KUKA KRL program: MyProgram_025().src

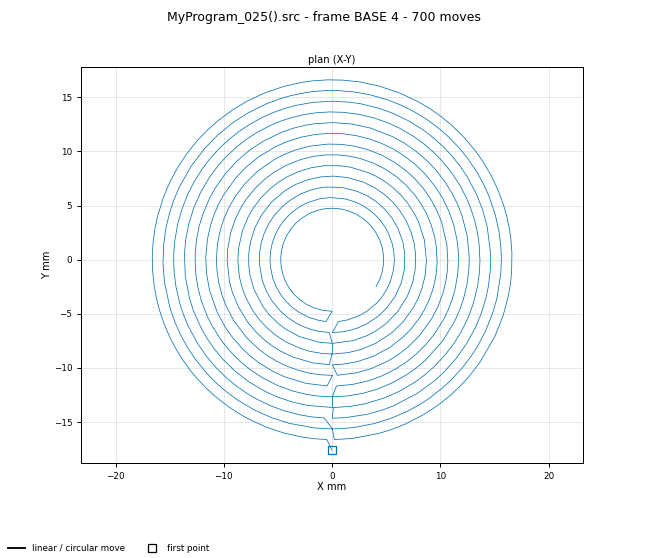
[picture p0: tool path of MyProgram_025().src in frame BASE 4, 700 of 700 moves have a stored position in this frame; points joined in program order, loops and branches not executed]
&ACCESS RVP
&REL 1
&PARAM TEMPLATE = C:\KRC\Roboter\Template\vorgabe
&PARAM EDITMASK = *
DEF MyProgram_025()
; ---- Setting reference (Base) ----
$BASE = BASE_DATA[4]

; --------------------------
; ---- Setting tool (TCP) ----
$TOOL = TOOL_DATA[3]
; --------------------------

$VEL.CP = VEL_APROX_PRINT
Startdeposition()
$VEL.CP = VEL_PRINT
LIN {X -0.0079,Y -17.5993,Z 57,A -96.7088,B 24.8277,C -3.0276,E1 25.0016,E2 -540.8331} C_DIS
Enddeposition()
LIN {X -0.0079,Y -17.5993,Z 57,A -96.7088,B 24.8277,C -3.0276,E1 25.0016,E2 -540.8331} C_DIS
Startdeposition()
$VEL.CP = VEL_PRINT
LIN {X -0.4966,Y -16.6086,Z 57,A -99.8681,B 24.8268,C -3.0359,E1 24.9929,E2 -537.6934} C_DIS
LIN {X -1.6135,Y -16.537,Z 57,A -103.5164,B 24.8266,C -3.0371,E1 24.9827,E2 -534.0464} C_DIS
LIN {X -2.8447,Y -16.3711,Z 57,A -108.4437,B 24.8269,C -3.0348,E1 24.9691,E2 -529.1094} C_DIS
LIN {X -4.4562,Y -16.0071,Z 57,A -114.0393,B 24.8265,C -3.0384,E1 24.9539,E2 -523.5144} C_DIS
LIN {X -6.0086,Y -15.4911,Z 57,A -120.3212,B 24.8262,C -3.0403,E1 24.9374,E2 -517.2245} C_DIS
LIN {X -7.613,Y -14.7693,Z 57,A -125.0534,B 24.8248,C -3.0528,E1 24.9255,E2 -512.51} C_DIS
LIN {X -8.4976,Y -14.2789,Z 57,A -129.0744,B 24.8245,C -3.0554,E1 24.9158,E2 -508.4833} C_DIS
LIN {X -9.6445,Y -13.5307,Z 57,A -134.1192,B 24.8238,C -3.0616,E1 24.9042,E2 -503.4363} C_DIS
LIN {X -10.8321,Y -12.6002,Z 57,A -138.7295,B 24.8225,C -3.073,E1 24.8942,E2 -498.8359} C_DIS
LIN {X -11.5957,Y -11.9014,Z 57,A -142.6614,B 24.8218,C -3.0788,E1 24.8862,E2 -494.9017} C_DIS
LIN {X -12.5279,Y -10.9156,Z 57,A -146.9241,B 24.8205,C -3.0901,E1 24.8782,E2 -490.6474} C_DIS
LIN {X -13.1346,Y -10.1775,Z 57,A -150.5821,B 24.8197,C -3.0966,E1 24.8718,E2 -486.9877} C_DIS
LIN {X -13.8252,Y -9.2175,Z 57,A -154.4634,B 24.8185,C -3.107,E1 24.8656,E2 -483.1122} C_DIS
LIN {X -14.4131,Y -8.2642,Z 57,A -158.3118,B 24.8173,C -3.117,E1 24.8601,E2 -479.2678} C_DIS
LIN {X -15.0085,Y -7.1299,Z 57,A -163.0011,B 24.816,C -3.128,E1 24.8542,E2 -474.5798} C_DIS
LIN {X -15.5303,Y -5.9078,Z 57,A -167.967,B 24.8146,C -3.1399,E1 24.849,E2 -469.6147} C_DIS
LIN {X -15.9455,Y -4.6722,Z 57,A -172.1158,B 24.813,C -3.1538,E1 24.8455,E2 -465.4753} C_DIS
LIN {X -16.2237,Y -3.5903,Z 57,A -175.9774,B 24.8116,C -3.1652,E1 24.843,E2 -461.6184} C_DIS
LIN {X -16.4274,Y -2.4984,Z 57,A -179.9383,B 24.8103,C -3.1765,E1 24.8412,E2 -457.6611} C_DIS
LIN {X -16.5879,Y -0.9632,Z 57,A 174.764,B 24.8083,C -3.1929,E1 24.8399,E2 -452.3709} C_DIS
LIN {X -16.6147,Y 0.2389,Z 57,A 170.0951,B 24.8069,C -3.2046,E1 24.8399,E2 -447.702} C_DIS
LIN {X -16.5377,Y 1.6093,Z 57,A 166.0881,B 24.8049,C -3.2209,E1 24.8407,E2 -443.71} C_DIS
LIN {X -16.379,Y 2.7981,Z 57,A 162.1452,B 24.8033,C -3.2342,E1 24.8423,E2 -439.7753} C_DIS
LIN {X -16.1488,Y 3.9123,Z 57,A 156.9096,B 24.8021,C -3.2434,E1 24.8455,E2 -434.531} C_DIS
LIN {X -15.6026,Y 5.7141,Z 57,A 150.5557,B 24.7997,C -3.2632,E1 24.8512,E2 -428.1884} C_DIS
LIN {X -15.0536,Y 7.0344,Z 57,A 145.873,B 24.7979,C -3.2781,E1 24.8565,E2 -423.5158} C_DIS
LIN {X -14.2835,Y 8.4901,Z 57,A 139.9499,B 24.7959,C -3.2935,E1 24.8645,E2 -417.5984} C_DIS
LIN {X -13.4224,Y 9.7912,Z 57,A 135.2799,B 24.7939,C -3.3097,E1 24.8719,E2 -412.9442} C_DIS
LIN {X -12.4942,Y 10.9541,Z 57,A 130.3829,B 24.7922,C -3.3233,E1 24.8806,E2 -408.057} C_DIS
LIN {X -11.6781,Y 11.8204,Z 57,A 125.1708,B 24.7914,C -3.3297,E1 24.8907,E2 -402.838} C_DIS
LIN {X -10.5248,Y 12.858,Z 57,A 120.5872,B 24.7896,C -3.3437,E1 24.9004,E2 -398.27} C_DIS
LIN {X -9.1848,Y 13.847,Z 57,A 114.2189,B 24.7885,C -3.3529,E1 24.9149,E2 -391.9016} C_DIS
LIN {X -7.7571,Y 14.6943,Z 57,A 108.4775,B 24.7873,C -3.3625,E1 24.9288,E2 -386.1666} C_DIS
LIN {X -6.1672,Y 15.429,Z 57,A 102.3711,B 24.7862,C -3.3708,E1 24.9445,E2 -380.0655} C_DIS
LIN {X -4.4893,Y 15.9979,Z 57,A 96.3662,B 24.7853,C -3.378,E1 24.9604,E2 -374.0674} C_DIS
LIN {X -2.884,Y 16.364,Z 57,A 90.9322,B 24.7846,C -3.3837,E1 24.9753,E2 -368.6406} C_DIS
LIN {X -1.7423,Y 16.5244,Z 57,A 86.9351,B 24.7843,C -3.3859,E1 24.9863,E2 -364.6459} C_DIS
LIN {X -0.406,Y 16.6112,Z 57,A 82.7039,B 24.7838,C -3.3894,E1 24.9981,E2 -360.422} C_DIS
LIN {X 0.9946,Y 16.5858,Z 57,A 77.1037,B 24.7843,C -3.3858,E1 25.0138,E2 -354.8146} C_DIS
LIN {X 2.6236,Y 16.4076,Z 57,A 71.2834,B 24.7846,C -3.3836,E1 25.0299,E2 -348.9939} C_DIS
LIN {X 4.2635,Y 16.0596,Z 57,A 65.3163,B 24.7851,C -3.3793,E1 25.046,E2 -343.0255} C_DIS
LIN {X 6.1988,Y 15.4163,Z 57,A 58.4682,B 24.7858,C -3.3743,E1 25.064,E2 -336.1796} C_DIS
LIN {X 8.0336,Y 14.5452,Z 57,A 52.1599,B 24.7863,C -3.3702,E1 25.0797,E2 -329.8788} C_DIS
LIN {X 8.9547,Y 13.9969,Z 57,A 48.0765,B 24.7873,C -3.3622,E1 25.0894,E2 -325.7892} C_DIS
LIN {X 10.1005,Y 13.1939,Z 57,A 43.99,B 24.7877,C -3.3593,E1 25.0986,E2 -321.7103} C_DIS
LIN {X 10.9536,Y 12.4947,Z 57,A 39.5699,B 24.7891,C -3.3478,E1 25.1081,E2 -317.28} C_DIS
LIN {X 12.0575,Y 11.4333,Z 57,A 34.1471,B 24.7906,C -3.3359,E1 25.1187,E2 -311.8518} C_DIS
LIN {X 13.1886,Y 10.1074,Z 57,A 29.0536,B 24.7915,C -3.3292,E1 25.1278,E2 -306.766} C_DIS
LIN {X 13.9189,Y 9.0749,Z 57,A 23.824,B 24.7937,C -3.3117,E1 25.136,E2 -301.5208} C_DIS
LIN {X 14.6967,Y 7.7524,Z 57,A 18.6399,B 24.7953,C -3.2987,E1 25.1431,E2 -296.3328} C_DIS
LIN {X 15.312,Y 6.4523,Z 57,A 14.2767,B 24.7964,C -3.2899,E1 25.1481,E2 -291.9724} C_DIS
LIN {X 15.8274,Y 5.0576,Z 57,A 8.8948,B 24.7985,C -3.2732,E1 25.1531,E2 -286.581} C_DIS
LIN {X 16.1435,Y 3.9343,Z 57,A 4.9444,B 24.7999,C -3.2619,E1 25.1559,E2 -282.6266} C_DIS
LIN {X 16.3628,Y 2.8911,Z 57,A 1.4471,B 24.801,C -3.2523,E1 25.1577,E2 -279.127} C_DIS
LIN {X 16.5081,Y 1.8912,Z 57,A -2.0127,B 24.8023,C -3.2418,E1 25.159,E2 -275.6629} C_DIS
LIN {X 16.6046,Y 0.6127,Z 57,A -7.3278,B 24.8049,C -3.2206,E1 25.1598,E2 -270.3291} C_DIS
LIN {X 16.572,Y -1.2047,Z 57,A -12.6063,B 24.8063,C -3.2095,E1 25.1592,E2 -265.0555} C_DIS
LIN {X 16.4651,Y -2.2352,Z 57,A -16.4567,B 24.8079,C -3.196,E1 25.1579,E2 -261.1959} C_DIS
LIN {X 16.2794,Y -3.328,Z 57,A -20.8494,B 24.8099,C -3.1794,E1 25.1555,E2 -256.7894} C_DIS
LIN {X 15.7843,Y -5.1905,Z 57,A -26.4474,B 24.8113,C -3.1679,E1 25.1512,E2 -251.1963} C_DIS
LIN {X 15.0304,Y -7.083,Z 57,A -35.0616,B 24.8153,C -3.1341,E1 25.1417,E2 -242.5491} C_DIS
LIN {X 13.6579,Y -9.4636,Z 57,A -44.0363,B 24.8179,C -3.1121,E1 25.1283,E2 -233.5676} C_DIS
LIN {X 12.6386,Y -10.7872,Z 57,A -48.808,B 24.8187,C -3.1052,E1 25.12,E2 -228.8016} C_DIS
LIN {X 11.8964,Y -11.6005,Z 57,A -52.9805,B 24.8201,C -3.0931,E1 25.1119,E2 -224.6186} C_DIS
LIN {X 10.9268,Y -12.5181,Z 57,A -57.6642,B 24.8214,C -3.0822,E1 25.1022,E2 -219.9277} C_DIS
LIN {X 9.7819,Y -13.4314,Z 57,A -62.0262,B 24.822,C -3.0768,E1 25.0925,E2 -215.569} C_DIS
LIN {X 8.4724,Y -14.2939,Z 57,A -68.8986,B 24.8244,C -3.0564,E1 25.0762,E2 -208.6699} C_DIS
LIN {X 6.7566,Y -15.18,Z 57,A -73.9115,B 24.8243,C -3.0574,E1 25.0636,E2 -203.6725} C_DIS
LIN {X 5.5988,Y -15.6442,Z 57,A -79.1554,B 24.8257,C -3.0455,E1 25.0499,E2 -198.4115} C_DIS
LIN {X 4.3439,Y -16.0381,Z 57,A -84.2086,B 24.8266,C -3.0374,E1 25.0363,E2 -193.3474} C_DIS
LIN {X 1.8661,Y -16.5109,Z 57,A -91.9923,B 24.8266,C -3.0367,E1 25.0148,E2 -185.5698} C_DIS
LIN {X 0.2013,Y -16.6148,Z 57,A -97.7093,B 24.8269,C -3.0348,E1 24.9989,E2 -179.85} C_DIS
LIN {X 0.2013,Y -16.6148,Z 57,A -97.7093,B 24.8269,C -3.0348,E1 24.9989,E2 -179.85} C_DIS
Enddeposition()
LIN {X 0.0206,Y -15.6269,Z 57,A -98.3842,B 24.8249,C -3.0519,E1 24.9971,E2 -179.2158} C_DIS
Startdeposition()
$VEL.CP = VEL_PRINT
LIN {X 0.9435,Y -15.599,Z 57,A -93.051,B 24.8236,C -3.0635,E1 25.0121,E2 -184.5756} C_DIS
LIN {X 2.0952,Y -15.4866,Z 57,A -87.9065,B 24.8227,C -3.0713,E1 25.0264,E2 -189.7346} C_DIS
LIN {X 3.9167,Y -15.1291,Z 57,A -81.5833,B 24.8223,C -3.0744,E1 25.0436,E2 -196.0569} C_DIS
LIN {X 5.5383,Y -14.6133,Z 57,A -74.7685,B 24.821,C -3.0859,E1 25.0616,E2 -202.8853} C_DIS
LIN {X 7.0237,Y -13.9605,Z 57,A -69.3589,B 24.8203,C -3.0913,E1 25.0752,E2 -208.2939} C_DIS
LIN {X 8.1308,Y -13.3463,Z 57,A -64.8305,B 24.8195,C -3.0987,E1 25.0862,E2 -212.826} C_DIS
LIN {X 8.9083,Y -12.8404,Z 57,A -61.1071,B 24.8184,C -3.1076,E1 25.0948,E2 -216.558} C_DIS
LIN {X 10.1325,Y -11.8962,Z 57,A -56.164,B 24.8176,C -3.1144,E1 25.1055,E2 -221.4985} C_DIS
LIN {X 10.9935,Y -11.1074,Z 57,A -51.3475,B 24.816,C -3.1283,E1 25.1153,E2 -226.328} C_DIS
LIN {X 11.9887,Y -10.0251,Z 57,A -46.5171,B 24.8149,C -3.1373,E1 25.1242,E2 -231.1582} C_DIS
LIN {X 12.7126,Y -9.0898,Z 57,A -41.7061,B 24.8131,C -3.1524,E1 25.1322,E2 -235.982} C_DIS
LIN {X 13.4007,Y -8.041,Z 57,A -37.5322,B 24.812,C -3.1617,E1 25.1384,E2 -240.1568} C_DIS
LIN {X 14.1741,Y -6.5816,Z 57,A -30.1128,B 24.8086,C -3.1903,E1 25.1476,E2 -247.6043} C_DIS
LIN {X 14.8853,Y -4.7586,Z 57,A -24.5547,B 24.8076,C -3.1984,E1 25.1529,E2 -253.1506} C_DIS
LIN {X 15.2207,Y -3.5422,Z 57,A -18.7319,B 24.8047,C -3.2226,E1 25.1568,E2 -258.9971} C_DIS
LIN {X 15.5726,Y -1.3083,Z 57,A -10.9381,B 24.802,C -3.2442,E1 25.1595,E2 -266.796} C_DIS
LIN {X 15.6284,Y 0.1312,Z 57,A -5.9472,B 24.8003,C -3.2581,E1 25.1597,E2 -271.7904} C_DIS
LIN {X 15.584,Y 1.1666,Z 57,A -2.2695,B 24.799,C -3.2689,E1 25.159,E2 -275.4717} C_DIS
LIN {X 15.4198,Y 2.542,Z 57,A 3.2023,B 24.7967,C -3.2876,E1 25.1568,E2 -280.9556} C_DIS
LIN {X 15.0687,Y 4.143,Z 57,A 9.0985,B 24.7946,C -3.3045,E1 25.1529,E2 -286.8578} C_DIS
LIN {X 14.4795,Y 5.8793,Z 57,A 14.6677,B 24.7933,C -3.3144,E1 25.1476,E2 -292.4193} C_DIS
LIN {X 14.0062,Y 6.932,Z 57,A 19.5498,B 24.7912,C -3.3311,E1 25.1418,E2 -297.3147} C_DIS
LIN {X 13.4124,Y 8.0215,Z 57,A 24.4658,B 24.7894,C -3.3457,E1 25.135,E2 -302.2399} C_DIS
LIN {X 12.4792,Y 9.4076,Z 57,A 29.473,B 24.7886,C -3.3521,E1 25.127,E2 -307.2378} C_DIS
LIN {X 11.77,Y 10.2811,Z 57,A 34.6706,B 24.7864,C -3.3693,E1 25.1176,E2 -312.4525} C_DIS
LIN {X 10.7719,Y 11.3227,Z 57,A 39.5954,B 24.7853,C -3.3775,E1 25.1079,E2 -317.376} C_DIS
LIN {X 9.7978,Y 12.1754,Z 57,A 44.5953,B 24.784,C -3.388,E1 25.0971,E2 -322.3816} C_DIS
LIN {X 8.7419,Y 12.9543,Z 57,A 49.3792,B 24.783,C -3.3956,E1 25.0862,E2 -327.1671} C_DIS
LIN {X 7.5454,Y 13.6859,Z 57,A 53.9445,B 24.7826,C -3.399,E1 25.0752,E2 -331.7266} C_DIS
LIN {X 6.4553,Y 14.232,Z 57,A 58.7039,B 24.7817,C -3.4061,E1 25.0632,E2 -336.4904} C_DIS
LIN {X 5.0645,Y 14.7843,Z 57,A 64.7046,B 24.7806,C -3.4141,E1 25.0475,E2 -342.4976} C_DIS
LIN {X 3.5259,Y 15.2249,Z 57,A 70.2952,B 24.7804,C -3.4159,E1 25.0324,E2 -348.0839} C_DIS
LIN {X 2.0313,Y 15.4953,Z 57,A 75.6659,B 24.7804,C -3.4164,E1 25.0175,E2 -353.4508} C_DIS
LIN {X 0.6375,Y 15.6142,Z 57,A 80.7731,B 24.7804,C -3.4164,E1 25.0033,E2 -358.5557} C_DIS
LIN {X -0.5666,Y 15.6174,Z 57,A 84.8908,B 24.7807,C -3.4138,E1 24.9918,E2 -362.6675} C_DIS
LIN {X -1.564,Y 15.5494,Z 57,A 88.6285,B 24.7808,C -3.4125,E1 24.9815,E2 -366.4039} C_DIS
LIN {X -2.3922,Y 15.4438,Z 57,A 92.0536,B 24.7808,C -3.4121,E1 24.972,E2 -369.831} C_DIS
LIN {X -3.8131,Y 15.1553,Z 57,A 97.2792,B 24.7815,C -3.4071,E1 24.9578,E2 -375.0513} C_DIS
LIN {X -4.8435,Y 14.858,Z 57,A 101.1242,B 24.7821,C -3.4024,E1 24.9475,E2 -378.8918} C_DIS
LIN {X -6.0233,Y 14.4203,Z 57,A 106.3248,B 24.7826,C -3.3985,E1 24.9341,E2 -384.0945} C_DIS
LIN {X -7.8381,Y 13.5204,Z 57,A 113.6192,B 24.7843,C -3.3859,E1 24.9161,E2 -391.3792} C_DIS
LIN {X -9.2432,Y 12.6012,Z 57,A 119.6077,B 24.7858,C -3.3736,E1 24.9024,E2 -397.3584} C_DIS
LIN {X -10.5413,Y 11.5372,Z 57,A 126.4152,B 24.7873,C -3.3621,E1 24.8881,E2 -404.1651} C_DIS
LIN {X -11.7783,Y 10.2715,Z 57,A 132.8456,B 24.7893,C -3.3462,E1 24.876,E2 -410.5859} C_DIS
LIN {X -13.0209,Y 8.6423,Z 57,A 140.7974,B 24.7917,C -3.3274,E1 24.8632,E2 -418.5316} C_DIS
LIN {X -14.1122,Y 6.7135,Z 57,A 147.5859,B 24.795,C -3.3013,E1 24.8543,E2 -425.2934} C_DIS
LIN {X -14.6037,Y 5.5642,Z 57,A 152.7773,B 24.7965,C -3.2891,E1 24.8489,E2 -430.4846} C_DIS
LIN {X -15.0043,Y 4.3697,Z 57,A 157.4172,B 24.7982,C -3.2751,E1 24.8451,E2 -435.1178} C_DIS
LIN {X -15.357,Y 2.8975,Z 57,A 162.3911,B 24.8005,C -3.2569,E1 24.8422,E2 -440.0771} C_DIS
LIN {X -15.5765,Y 1.2631,Z 57,A 168.5705,B 24.8028,C -3.2384,E1 24.8401,E2 -446.2491} C_DIS
LIN {X -15.6241,Y -0.329,Z 57,A 175.0512,B 24.8048,C -3.2215,E1 24.84,E2 -452.7286} C_DIS
LIN {X -15.4932,Y -2.0432,Z 57,A -177.8917,B 24.807,C -3.2039,E1 24.8421,E2 -459.7855} C_DIS
LIN {X -14.9848,Y -4.4352,Z 57,A -169.1992,B 24.8102,C -3.1767,E1 24.848,E2 -468.4636} C_DIS
LIN {X -14.5084,Y -5.8074,Z 57,A -164.7835,B 24.8123,C -3.1595,E1 24.8523,E2 -472.8629} C_DIS
LIN {X -13.9987,Y -6.9471,Z 57,A -159.8629,B 24.8137,C -3.1478,E1 24.8581,E2 -477.7825} C_DIS
LIN {X -13.3271,Y -8.1622,Z 57,A -155.194,B 24.8154,C -3.1336,E1 24.8646,E2 -482.4416} C_DIS
LIN {X -12.6612,Y -9.1613,Z 57,A -150.6238,B 24.8166,C -3.1233,E1 24.8718,E2 -487.0098} C_DIS
LIN {X -11.5607,Y -10.5159,Z 57,A -143.9703,B 24.8182,C -3.1098,E1 24.8838,E2 -493.6614} C_DIS
LIN {X -10.7026,Y -11.3881,Z 57,A -139.3705,B 24.8192,C -3.1011,E1 24.893,E2 -498.2597} C_DIS
LIN {X -9.7596,Y -12.206,Z 57,A -134.458,B 24.82,C -3.094,E1 24.9036,E2 -503.1738} C_DIS
LIN {X -8.6811,Y -12.9951,Z 57,A -129.5705,B 24.8209,C -3.0862,E1 24.9148,E2 -508.0593} C_DIS
LIN {X -7.2158,Y -13.8623,Z 57,A -123.6356,B 24.822,C -3.0767,E1 24.9292,E2 -513.9887} C_DIS
LIN {X -5.6053,Y -14.5873,Z 57,A -116.862,B 24.8226,C -3.0715,E1 24.9466,E2 -520.7655} C_DIS
LIN {X -3.9344,Y -15.1237,Z 57,A -109.7797,B 24.8228,C -3.0703,E1 24.9657,E2 -527.8565} C_DIS
LIN {X -1.6167,Y -15.5433,Z 57,A -101.5452,B 24.8232,C -3.0663,E1 24.9884,E2 -536.0883} C_DIS
LIN {X 0.0206,Y -15.6269,Z 57,A -98.3841,B 24.8249,C -3.0519,E1 24.9971,E2 -539.2158} C_DIS
Enddeposition()
LIN {X 0.0206,Y -15.6269,Z 57,A -98.3841,B 24.8249,C -3.0519,E1 24.9971,E2 -539.2158} C_DIS
Startdeposition()
$VEL.CP = VEL_PRINT
LIN {X -0.727,Y -14.6201,Z 57,A -99.9282,B 24.8222,C -3.0758,E1 24.993,E2 -537.7283} C_DIS
LIN {X -1.8741,Y -14.519,Z 57,A -105.7448,B 24.8228,C -3.07,E1 24.9767,E2 -531.8947} C_DIS
LIN {X -2.9932,Y -14.3301,Z 57,A -110.624,B 24.8228,C -3.0697,E1 24.9634,E2 -527.0095} C_DIS
LIN {X -4.5052,Y -13.929,Z 57,A -116.4703,B 24.8223,C -3.0748,E1 24.9477,E2 -521.1658} C_DIS
LIN {X -5.7524,Y -13.4618,Z 57,A -121.1932,B 24.8215,C -3.0815,E1 24.9354,E2 -516.4487} C_DIS
LIN {X -6.9719,Y -12.8729,Z 57,A -126.8563,B 24.8209,C -3.0865,E1 24.9213,E2 -510.7825} C_DIS
LIN {X -7.8805,Y -12.3378,Z 57,A -130.967,B 24.8202,C -3.0925,E1 24.9115,E2 -506.6734} C_DIS
LIN {X -8.8659,Y -11.65,Z 57,A -136.0466,B 24.8194,C -3.0992,E1 24.9001,E2 -501.5918} C_DIS
LIN {X -9.8302,Y -10.8484,Z 57,A -141.0341,B 24.8184,C -3.1082,E1 24.8896,E2 -496.6061} C_DIS
LIN {X -10.7742,Y -9.9116,Z 57,A -145.9486,B 24.817,C -3.1198,E1 24.8801,E2 -491.6982} C_DIS
LIN {X -11.6093,Y -8.9188,Z 57,A -150.7478,B 24.8156,C -3.132,E1 24.8717,E2 -486.9058} C_DIS
LIN {X -12.4595,Y -7.6864,Z 57,A -157.46,B 24.8141,C -3.1446,E1 24.8614,E2 -480.1903} C_DIS
LIN {X -13.3123,Y -6.091,Z 57,A -163.7129,B 24.8116,C -3.1652,E1 24.8535,E2 -473.9531} C_DIS
LIN {X -13.7409,Y -5.0496,Z 57,A -168.4392,B 24.8102,C -3.177,E1 24.8486,E2 -469.2286} C_DIS
LIN {X -14.0821,Y -4.0011,Z 57,A -172.8713,B 24.8087,C -3.1893,E1 24.8451,E2 -464.8005} C_DIS
LIN {X -14.427,Y -2.4862,Z 57,A -178.9816,B 24.8065,C -3.2075,E1 24.8416,E2 -458.6978} C_DIS
LIN {X -14.5795,Y -1.3229,Z 57,A 176.5908,B 24.8048,C -3.2218,E1 24.8402,E2 -454.278} C_DIS
LIN {X -14.6359,Y -0.3226,Z 57,A 172.6371,B 24.8033,C -3.2339,E1 24.8398,E2 -450.3294} C_DIS
LIN {X -14.6214,Y 0.7252,Z 57,A 168.6853,B 24.8017,C -3.2468,E1 24.8401,E2 -446.3849} C_DIS
LIN {X -14.5253,Y 1.8271,Z 57,A 164.1215,B 24.8001,C -3.2599,E1 24.8414,E2 -441.8251} C_DIS
LIN {X -14.2573,Y 3.3241,Z 57,A 157.8504,B 24.7979,C -3.2778,E1 24.8448,E2 -435.5598} C_DIS
LIN {X -13.8804,Y 4.6525,Z 57,A 152.7161,B 24.7958,C -3.2946,E1 24.849,E2 -430.4362} C_DIS
LIN {X -13.3302,Y 6.0517,Z 57,A 146.6742,B 24.7937,C -3.3116,E1 24.8554,E2 -424.4016} C_DIS
LIN {X -12.7704,Y 7.1581,Z 57,A 141.3649,B 24.7921,C -3.3245,E1 24.8624,E2 -419.0951} C_DIS
LIN {X -12.0193,Y 8.3581,Z 57,A 136.3567,B 24.79,C -3.3405,E1 24.87,E2 -414.1001} C_DIS
LIN {X -11.3764,Y 9.2141,Z 57,A 131.6096,B 24.7888,C -3.3501,E1 24.8782,E2 -409.3535} C_DIS
LIN {X -10.4642,Y 10.2384,Z 57,A 127.0245,B 24.787,C -3.3648,E1 24.8868,E2 -404.7834} C_DIS
LIN {X -9.6594,Y 11.0006,Z 57,A 121.9356,B 24.786,C -3.3727,E1 24.8973,E2 -399.6929} C_DIS
LIN {X -8.7045,Y 11.7707,Z 57,A 116.9211,B 24.7848,C -3.382,E1 24.9084,E2 -394.6823} C_DIS
LIN {X -7.7071,Y 12.4469,Z 57,A 112.2248,B 24.7837,C -3.3907,E1 24.9194,E2 -389.9918} C_DIS
LIN {X -6.4486,Y 13.1427,Z 57,A 106.7525,B 24.7824,C -3.4002,E1 24.933,E2 -384.5272} C_DIS
LIN {X -5.475,Y 13.577,Z 57,A 102.5199,B 24.7817,C -3.4057,E1 24.9438,E2 -380.2983} C_DIS
LIN {X -4.3377,Y 13.9821,Z 57,A 98.2789,B 24.7808,C -3.4129,E1 24.9551,E2 -376.0664} C_DIS
LIN {X -3.2931,Y 14.2626,Z 57,A 94.0578,B 24.7803,C -3.417,E1 24.9665,E2 -371.8491} C_DIS
LIN {X -1.7846,Y 14.5305,Z 57,A 86.814,B 24.7803,C -3.416,E1 24.9865,E2 -364.5966} C_DIS
LIN {X 0.1204,Y 14.6392,Z 57,A 79.8797,B 24.7798,C -3.4203,E1 25.0058,E2 -357.6719} C_DIS
LIN {X 1.7666,Y 14.5325,Z 57,A 73.5904,B 24.7798,C -3.4205,E1 25.0233,E2 -351.3868} C_DIS
LIN {X 2.6817,Y 14.3921,Z 57,A 69.5206,B 24.7803,C -3.417,E1 25.0345,E2 -347.313} C_DIS
LIN {X 4.3798,Y 13.9686,Z 57,A 63.3585,B 24.7803,C -3.4162,E1 25.051,E2 -341.1592} C_DIS
LIN {X 5.5219,Y 13.5581,Z 57,A 58.7719,B 24.7808,C -3.4128,E1 25.063,E2 -336.5742} C_DIS
LIN {X 7.0572,Y 12.8266,Z 57,A 51.5599,B 24.7823,C -3.4014,E1 25.081,E2 -329.3547} C_DIS
LIN {X 8.2835,Y 12.0709,Z 57,A 46.4058,B 24.783,C -3.3958,E1 25.093,E2 -324.2041} C_DIS
LIN {X 9.0887,Y 11.4768,Z 57,A 42.1889,B 24.7841,C -3.387,E1 25.1024,E2 -319.9818} C_DIS
LIN {X 10.1918,Y 10.5096,Z 57,A 36.5859,B 24.7854,C -3.3767,E1 25.1139,E2 -314.3771} C_DIS
LIN {X 11.0864,Y 9.5572,Z 57,A 31.9136,B 24.7865,C -3.3687,E1 25.1227,E2 -309.7065} C_DIS
LIN {X 11.7691,Y 8.707,Z 57,A 27.2705,B 24.7881,C -3.3561,E1 25.1306,E2 -305.0553} C_DIS
LIN {X 12.4611,Y 7.6842,Z 57,A 22.0827,B 24.7899,C -3.3414,E1 25.1384,E2 -299.8588} C_DIS
LIN {X 13.3557,Y 5.9948,Z 57,A 15.3741,B 24.7917,C -3.3271,E1 25.1468,E2 -293.1519} C_DIS
LIN {X 13.8737,Y 4.6711,Z 57,A 9.2407,B 24.7943,C -3.307,E1 25.1527,E2 -287.0051} C_DIS
LIN {X 14.3243,Y 3.0191,Z 57,A 1.7255,B 24.7975,C -3.2809,E1 25.1576,E2 -279.4715} C_DIS
LIN {X 14.626,Y 0.6192,Z 57,A -6.9873,B 24.8004,C -3.2576,E1 25.1598,E2 -270.7551} C_DIS
LIN {X 14.6121,Y -0.8882,Z 57,A -12.9408,B 24.8027,C -3.2388,E1 25.1591,E2 -264.7925} C_DIS
LIN {X 14.4336,Y -2.4485,Z 57,A -18.4748,B 24.8045,C -3.2245,E1 25.157,E2 -259.2571} C_DIS
LIN {X 14.2046,Y -3.5403,Z 57,A -22.5259,B 24.8058,C -3.2135,E1 25.1544,E2 -255.2034} C_DIS
LIN {X 13.7439,Y -5.0418,Z 57,A -28.8614,B 24.8082,C -3.1934,E1 25.1489,E2 -248.8564} C_DIS
LIN {X 13.2317,Y -6.264,Z 57,A -34.2216,B 24.8102,C -3.1769,E1 25.1429,E2 -243.4861} C_DIS
LIN {X 12.4157,Y -7.7565,Z 57,A -41.7381,B 24.8132,C -3.152,E1 25.1322,E2 -235.9491} C_DIS
LIN {X 11.4139,Y -9.1679,Z 57,A -47.6621,B 24.8146,C -3.1405,E1 25.1222,E2 -230.0259} C_DIS
LIN {X 10.2913,Y -10.412,Z 57,A -53.7451,B 24.816,C -3.128,E1 25.1106,E2 -223.94} C_DIS
LIN {X 9.4715,Y -11.1631,Z 57,A -58.7876,B 24.8177,C -3.1136,E1 25.0999,E2 -218.8831} C_DIS
LIN {X 7.8982,Y -12.3264,Z 57,A -67.3187,B 24.8201,C -3.093,E1 25.0802,E2 -210.3321} C_DIS
LIN {X 5.7082,Y -13.4806,Z 57,A -75.3487,B 24.8207,C -3.0882,E1 25.0601,E2 -202.3119} C_DIS
LIN {X 4.7288,Y -13.8548,Z 57,A -79.7629,B 24.8215,C -3.0812,E1 25.0485,E2 -197.8901} C_DIS
LIN {X 3.1832,Y -14.2895,Z 57,A -86.9746,B 24.8228,C -3.0698,E1 25.0289,E2 -190.662} C_DIS
LIN {X 1.1917,Y -14.5909,Z 57,A -93.7861,B 24.8228,C -3.0708,E1 25.0101,E2 -183.858} C_DIS
LIN {X 0.0018,Y -14.6384,Z 57,A -96.216,B 24.8216,C -3.0806,E1 25.0034,E2 -181.4522} C_DIS
Enddeposition()
LIN {X 0.0018,Y -14.6384,Z 57,A -96.216,B 24.8216,C -3.0806,E1 25.0034,E2 -181.4522} C_DIS
Startdeposition()
$VEL.CP = VEL_PRINT
LIN {X 0.1135,Y -13.6506,Z 57,A -94.9951,B 24.8192,C -3.1012,E1 25.0069,E2 -182.7218} C_DIS
LIN {X 1.5958,Y -13.5576,Z 57,A -89.274,B 24.8192,C -3.1017,E1 25.0228,E2 -188.4409} C_DIS
LIN {X 3.0042,Y -13.3167,Z 57,A -82.7157,B 24.8182,C -3.1098,E1 25.0408,E2 -195.0103} C_DIS
LIN {X 4.8633,Y -12.7557,Z 57,A -76.029,B 24.818,C -3.111,E1 25.0585,E2 -201.6873} C_DIS
LIN {X 6.2683,Y -12.1269,Z 57,A -67.756,B 24.8156,C -3.132,E1 25.0794,E2 -209.9887} C_DIS
LIN {X 7.6568,Y -11.302,Z 57,A -62.1769,B 24.815,C -3.1369,E1 25.0925,E2 -215.5614} C_DIS
LIN {X 8.5156,Y -10.67,Z 57,A -57.6116,B 24.8138,C -3.1467,E1 25.1026,E2 -220.1334} C_DIS
LIN {X 9.4267,Y -9.8742,Z 57,A -52.1979,B 24.8122,C -3.1606,E1 25.1138,E2 -225.5579} C_DIS
LIN {X 10.4265,Y -8.8079,Z 57,A -46.8243,B 24.811,C -3.1703,E1 25.1238,E2 -230.9309} C_DIS
LIN {X 11.2741,Y -7.698,Z 57,A -40.3869,B 24.8086,C -3.1899,E1 25.1344,E2 -237.3836} C_DIS
LIN {X 11.9086,Y -6.6743,Z 57,A -35.2024,B 24.8068,C -3.205,E1 25.1417,E2 -242.5772} C_DIS
LIN {X 12.5448,Y -5.3837,Z 57,A -29.797,B 24.8053,C -3.2179,E1 25.148,E2 -247.9838} C_DIS
LIN {X 13.0399,Y -4.0393,Z 57,A -23.0076,B 24.8023,C -3.2419,E1 25.1541,E2 -254.7919} C_DIS
LIN {X 13.4264,Y -2.4692,Z 57,A -16.7624,B 24.8003,C -3.2586,E1 25.1578,E2 -261.0404} C_DIS
LIN {X 13.6038,Y -1.1366,Z 57,A -11.6238,B 24.7986,C -3.2723,E1 25.1594,E2 -266.1811} C_DIS
LIN {X 13.6523,Y -0.0889,Z 57,A -7.0772,B 24.7967,C -3.2871,E1 25.1598,E2 -270.7358} C_DIS
LIN {X 13.5801,Y 1.3936,Z 57,A -0.7639,B 24.7943,C -3.307,E1 25.1586,E2 -277.0587} C_DIS
LIN {X 13.4093,Y 2.5598,Z 57,A 4.2838,B 24.7923,C -3.3227,E1 25.1562,E2 -282.1141} C_DIS
LIN {X 13.1622,Y 3.6214,Z 57,A 8.5349,B 24.7909,C -3.3338,E1 25.1533,E2 -286.367} C_DIS
LIN {X 12.8062,Y 4.7199,Z 57,A 13.2193,B 24.7893,C -3.3466,E1 25.149,E2 -291.0553} C_DIS
LIN {X 12.3941,Y 5.7221,Z 57,A 18.2123,B 24.7873,C -3.3624,E1 25.1434,E2 -296.0584} C_DIS
LIN {X 11.8129,Y 6.8425,Z 57,A 23.3194,B 24.7857,C -3.3749,E1 25.1365,E2 -301.1686} C_DIS
LIN {X 11.0579,Y 8.0054,Z 57,A 29.2785,B 24.7837,C -3.3901,E1 25.1272,E2 -307.1345} C_DIS
LIN {X 10.1702,Y 9.1066,Z 57,A 35.2885,B 24.782,C -3.4039,E1 25.1163,E2 -313.1498} C_DIS
LIN {X 9.3437,Y 9.9528,Z 57,A 39.7727,B 24.7811,C -3.4108,E1 25.1073,E2 -317.6317} C_DIS
LIN {X 8.4234,Y 10.743,Z 57,A 45.0195,B 24.7797,C -3.4211,E1 25.096,E2 -322.8828} C_DIS
LIN {X 7.4952,Y 11.4099,Z 57,A 49.9876,B 24.7786,C -3.4297,E1 25.0846,E2 -327.8546} C_DIS
LIN {X 6.2545,Y 12.1341,Z 57,A 55.992,B 24.7776,C -3.4376,E1 25.0699,E2 -333.8603} C_DIS
LIN {X 5.1835,Y 12.6291,Z 57,A 60.8874,B 24.777,C -3.4425,E1 25.0573,E2 -338.7556} C_DIS
LIN {X 3.8204,Y 13.1057,Z 57,A 67.2511,B 24.7761,C -3.4487,E1 25.0404,E2 -345.1222} C_DIS
LIN {X 2.4098,Y 13.4371,Z 57,A 72.9463,B 24.7761,C -3.4494,E1 25.0249,E2 -350.8121} C_DIS
LIN {X 1.029,Y 13.6124,Z 57,A 79.001,B 24.7758,C -3.4511,E1 25.008,E2 -356.867} C_DIS
LIN {X -0.2481,Y 13.6491,Z 57,A 84.1645,B 24.7761,C -3.4493,E1 24.9936,E2 -362.0258} C_DIS
LIN {X -1.5088,Y 13.5657,Z 57,A 89.1148,B 24.7766,C -3.4455,E1 24.9799,E2 -366.9694} C_DIS
LIN {X -2.6162,Y 13.3985,Z 57,A 94.4185,B 24.7767,C -3.4443,E1 24.9653,E2 -372.2756} C_DIS
LIN {X -3.9193,Y 13.0747,Z 57,A 99.4222,B 24.7777,C -3.4366,E1 24.9518,E2 -377.2683} C_DIS
LIN {X -4.7015,Y 12.8137,Z 57,A 102.9102,B 24.7783,C -3.4325,E1 24.9427,E2 -380.7534} C_DIS
LIN {X -5.656,Y 12.4245,Z 57,A 107.8676,B 24.7788,C -3.4283,E1 24.93,E2 -385.7124} C_DIS
LIN {X -6.903,Y 11.7777,Z 57,A 113.7791,B 24.7801,C -3.4185,E1 24.9155,E2 -391.6174} C_DIS
LIN {X -7.8374,Y 11.1775,Z 57,A 118.4241,B 24.7812,C -3.4095,E1 24.9048,E2 -396.2566} C_DIS
LIN {X -8.7366,Y 10.4898,Z 57,A 123.0958,B 24.7825,C -3.3994,E1 24.8947,E2 -400.9215} C_DIS
LIN {X -9.8197,Y 9.4835,Z 57,A 129.1177,B 24.7844,C -3.3847,E1 24.8827,E2 -406.9334} C_DIS
LIN {X -10.5398,Y 8.6757,Z 57,A 133.8788,B 24.7858,C -3.3739,E1 24.874,E2 -411.6902} C_DIS
LIN {X -11.3068,Y 7.6498,Z 57,A 139.3398,B 24.7876,C -3.3598,E1 24.8652,E2 -417.1443} C_DIS
LIN {X -12.0845,Y 6.3503,Z 57,A 146.0981,B 24.7898,C -3.3427,E1 24.856,E2 -423.8969} C_DIS
LIN {X -12.7902,Y 4.7713,Z 57,A 152.0093,B 24.7927,C -3.3194,E1 24.8496,E2 -429.7849} C_DIS
LIN {X -13.2544,Y 3.2578,Z 57,A 159.3523,B 24.7951,C -3.3002,E1 24.8438,E2 -437.1244} C_DIS
LIN {X -13.5257,Y 1.8494,Z 57,A 165.9926,B 24.7973,C -3.2824,E1 24.8407,E2 -443.7614} C_DIS
LIN {X -13.6401,Y 0.5494,Z 57,A 171.897,B 24.7994,C -3.266,E1 24.8398,E2 -449.662} C_DIS
LIN {X -13.5682,Y -1.5041,Z 57,A -178.9141,B 24.8025,C -3.2403,E1 24.8417,E2 -458.8444} C_DIS
LIN {X -13.1637,Y -3.6161,Z 57,A -171.3042,B 24.8061,C -3.2112,E1 24.8463,E2 -466.4292} C_DIS
LIN {X -12.7951,Y -4.7582,Z 57,A -165.2018,B 24.8076,C -3.1986,E1 24.8519,E2 -472.536} C_DIS
LIN {X -12.0262,Y -6.4602,Z 57,A -157.7712,B 24.8102,C -3.1767,E1 24.861,E2 -479.9543} C_DIS
LIN {X -11.5485,Y -7.2799,Z 57,A -154.0085,B 24.8115,C -3.1662,E1 24.8665,E2 -483.7111} C_DIS
LIN {X -10.8381,Y -8.3006,Z 57,A -148.9133,B 24.813,C -3.1535,E1 24.8749,E2 -488.8006} C_DIS
LIN {X -10.0592,Y -9.2291,Z 57,A -143.5583,B 24.8143,C -3.143,E1 24.8847,E2 -494.1546} C_DIS
LIN {X -8.9517,Y -10.3069,Z 57,A -136.6012,B 24.8156,C -3.1316,E1 24.899,E2 -501.1127} C_DIS
LIN {X -7.6898,Y -11.2795,Z 57,A -129.6655,B 24.8168,C -3.1214,E1 24.9148,E2 -508.0482} C_DIS
LIN {X -6.1325,Y -12.1965,Z 57,A -122.7827,B 24.8182,C -3.1093,E1 24.9316,E2 -514.9217} C_DIS
LIN {X -4.9876,Y -12.7073,Z 57,A -117.8834,B 24.819,C -3.1027,E1 24.9441,E2 -519.8166} C_DIS
LIN {X -3.6553,Y -13.1526,Z 57,A -111.8732,B 24.8195,C -3.0989,E1 24.9602,E2 -525.8283} C_DIS
LIN {X -2.2509,Y -13.4645,Z 57,A -104.3244,B 24.819,C -3.1031,E1 24.9809,E2 -533.3953} C_DIS
LIN {X 0.0359,Y -13.648,Z 57,A -99.2824,B 24.8214,C -3.0825,E1 24.9948,E2 -538.3904} C_DIS
Enddeposition()
LIN {X 0.0193,Y -12.6632,Z 57,A -3.1817,B 0,C 0,E1 0.1598,E2 -629.9291} C_DIS
Startdeposition()
$VEL.CP = VEL_PRINT
LIN {X -1.2428,Y -12.6019,Z 57,A -3.2256,B 0,C 0,E1 0.1598,E2 -629.9288} C_DIS
LIN {X -2.3509,Y -12.4426,Z 57,A -3.2593,B 0,C 0,E1 0.1598,E2 -629.9288} C_DIS
LIN {X -3.5963,Y -12.1416,Z 57,A -3.292,B 0,C 0,E1 0.1598,E2 -629.9288} C_DIS
LIN {X -5.0475,Y -11.6135,Z 57,A -3.3224,B 0,C 0,E1 0.1598,E2 -629.9291} C_DIS
LIN {X -6.4054,Y -10.9209,Z 57,A -3.3426,B 0,C 0,E1 0.1598,E2 -629.9291} C_DIS
LIN {X -7.532,Y -10.1799,Z 57,A -3.3523,B 0,C 0,E1 0.1598,E2 -629.9292} C_DIS
LIN {X -8.3604,Y -9.5112,Z 57,A -3.3542,B 0,C 0,E1 0.1598,E2 -629.9292} C_DIS
LIN {X -9.3471,Y -8.5434,Z 57,A -3.349,B 0,C 0,E1 0.1598,E2 -629.9294} C_DIS
LIN {X -10.1798,Y -7.5322,Z 57,A -3.3366,B 0,C 0,E1 0.1598,E2 -629.9294} C_DIS
LIN {X -11.0457,Y -6.1928,Z 57,A -3.3112,B 0,C 0,E1 0.1598,E2 -629.9297} C_DIS
LIN {X -11.4776,Y -5.3495,Z 57,A -3.2915,B 0,C 0,E1 0.1598,E2 -629.9295} C_DIS
LIN {X -12.0761,Y -3.8104,Z 57,A -3.2475,B 0,C 0,E1 0.1598,E2 -629.9302} C_DIS
LIN {X -12.3926,Y -2.5999,Z 57,A -3.2085,B 0,C 0,E1 0.1598,E2 -629.9295} C_DIS
LIN {X -12.5695,Y -1.5374,Z 57,A -3.1701,B 0,C 0,E1 0.1598,E2 -629.9294} C_DIS
LIN {X -12.6419,Y -0.7252,Z 57,A -3.1388,B 0,C 0,E1 0.1598,E2 -629.9289} C_DIS
LIN {X -12.6524,Y 0.518,Z 57,A -3.0861,B 0,C 0,E1 0.1598,E2 -629.9294} C_DIS
LIN {X -12.5243,Y 1.8718,Z 57,A -3.0241,B 0,C 0,E1 0.1598,E2 -629.9294} C_DIS
LIN {X -12.2883,Y 3.058,Z 57,A -2.9654,B 0,C 0,E1 0.1598,E2 -629.9292} C_DIS
LIN {X -11.964,Y 4.1488,Z 57,A -2.9074,B 0,C 0,E1 0.1598,E2 -629.929} C_DIS
LIN {X -11.3142,Y 5.6867,Z 57,A -2.8178,B 0,C 0,E1 0.1598,E2 -629.9295} C_DIS
LIN {X -10.7726,Y 6.6564,Z 57,A -2.7577,B 0,C 0,E1 0.1598,E2 -629.9286} C_DIS
LIN {X -9.8335,Y 7.9786,Z 57,A -2.6668,B 0,C 0,E1 0.1598,E2 -629.9288} C_DIS
LIN {X -8.8343,Y 9.0729,Z 57,A -2.5837,B 0,C 0,E1 0.1598,E2 -629.9287} C_DIS
LIN {X -7.6944,Y 10.0576,Z 57,A -2.5003,B 0,C 0,E1 0.1598,E2 -629.9282} C_DIS
LIN {X -6.4888,Y 10.8744,Z 57,A -2.4212,B 0,C 0,E1 0.1598,E2 -629.9282} C_DIS
LIN {X -4.7388,Y 11.7428,Z 57,A -2.3198,B 0,C 0,E1 0.1598,E2 -629.9279} C_DIS
LIN {X -3.5589,Y 12.1526,Z 57,A -2.2591,B 0,C 0,E1 0.1598,E2 -629.9275} C_DIS
LIN {X -2.5167,Y 12.4106,Z 57,A -2.2097,B 0,C 0,E1 0.1598,E2 -629.9275} C_DIS
LIN {X -1.5665,Y 12.5661,Z 57,A -2.168,B 0,C 0,E1 0.1598,E2 -629.9273} C_DIS
LIN {X 0.1656,Y 12.6621,Z 57,A -2.0998,B 0,C 0,E1 0.1598,E2 -629.9273} C_DIS
LIN {X 1.8294,Y 12.53,Z 57,A -2.0438,B 0,C 0,E1 0.1598,E2 -629.9272} C_DIS
LIN {X 3.5329,Y 12.1596,Z 57,A -1.9965,B 0,C 0,E1 0.1598,E2 -629.9272} C_DIS
LIN {X 5.5471,Y 11.3834,Z 57,A -1.9548,B 0,C 0,E1 0.1598,E2 -629.9274} C_DIS
LIN {X 6.6973,Y 10.7473,Z 57,A -1.9395,B 0,C 0,E1 0.1598,E2 -629.9274} C_DIS
LIN {X 7.7623,Y 10.0053,Z 57,A -1.9317,B 0,C 0,E1 0.1598,E2 -629.9274} C_DIS
LIN {X 8.8051,Y 9.101,Z 57,A -1.9316,B 0,C 0,E1 0.1598,E2 -629.9276} C_DIS
LIN {X 9.5098,Y 8.3616,Z 57,A -1.9374,B 0,C 0,E1 0.1598,E2 -629.9274} C_DIS
LIN {X 10.4439,Y 7.1613,Z 57,A -1.9535,B 0,C 0,E1 0.1598,E2 -629.928} C_DIS
LIN {X 11.1344,Y 6.0318,Z 57,A -1.9766,B 0,C 0,E1 0.1598,E2 -629.9278} C_DIS
LIN {X 11.564,Y 5.1598,Z 57,A -1.9983,B 0,C 0,E1 0.1598,E2 -629.9276} C_DIS
LIN {X 11.998,Y 4.0496,Z 57,A -2.0297,B 0,C 0,E1 0.1598,E2 -629.9278} C_DIS
LIN {X 12.4773,Y 2.1621,Z 57,A -2.0916,B 0,C 0,E1 0.1598,E2 -629.9292} C_DIS
LIN {X 12.6621,Y 0.1864,Z 57,A -2.1688,B 0,C 0,E1 0.1598,E2 -629.9299} C_DIS
LIN {X 12.6621,Y 0.1864,Z 57,A -2.1701,B 0,C 0,E1 0.1598,E2 -629.9286} C_DIS
LIN {X 12.6307,Y -0.8732,Z 57,A -2.2173,B 0,C 0,E1 0.1598,E2 -629.9281} C_DIS
LIN {X 12.4687,Y -2.2114,Z 57,A -2.2803,B 0,C 0,E1 0.1598,E2 -629.9285} C_DIS
LIN {X 12.1209,Y -3.6651,Z 57,A -2.3553,B 0,C 0,E1 0.1598,E2 -629.9287} C_DIS
LIN {X 11.7787,Y -4.6491,Z 57,A -2.4103,B 0,C 0,E1 0.1598,E2 -629.9287} C_DIS
LIN {X 11.2852,Y -5.7445,Z 57,A -2.4757,B 0,C 0,E1 0.1598,E2 -629.9284} C_DIS
LIN {X 10.1926,Y -7.5148,Z 57,A -2.5907,B 0,C 0,E1 0.1598,E2 -629.9296} C_DIS
LIN {X 8.6301,Y -9.267,Z 57,A -2.7239,B 0,C 0,E1 0.1598,E2 -629.9288} C_DIS
LIN {X 7.8114,Y -9.9668,Z 57,A -2.7843,B 0,C 0,E1 0.1598,E2 -629.9285} C_DIS
LIN {X 7.0205,Y -10.5388,Z 57,A -2.838,B 0,C 0,E1 0.1598,E2 -629.9284} C_DIS
LIN {X 5.6264,Y -11.3444,Z 57,A -2.9235,B 0,C 0,E1 0.1598,E2 -629.9285} C_DIS
LIN {X 4.1816,Y -11.9526,Z 57,A -3.0024,B 0,C 0,E1 0.1598,E2 -629.9285} C_DIS
LIN {X 2.8252,Y -12.3439,Z 57,A -3.0688,B 0,C 0,E1 0.1598,E2 -629.9285} C_DIS
LIN {X 1.3475,Y -12.5907,Z 57,A -3.1335,B 0,C 0,E1 0.1598,E2 -629.9286} C_DIS
LIN {X 0.0193,Y -12.6632,Z 57,A -3.1852,B 0,C 0,E1 0.1598,E2 -629.9286} C_DIS
Enddeposition()
LIN {X 0.0193,Y -12.6632,Z 57,A -3.1852,B 0,C 0,E1 0.1598,E2 -629.9286} C_DIS
Startdeposition()
$VEL.CP = VEL_PRINT
LIN {X 0.3938,Y -11.668,Z 57,A -3.128,B 0,C 0,E1 0.1598,E2 -629.9293} C_DIS
LIN {X 1.881,Y -11.5226,Z 57,A -3.0679,B 0,C 0,E1 0.1598,E2 -629.9286} C_DIS
LIN {X 3.381,Y -11.1742,Z 57,A -2.9981,B 0,C 0,E1 0.1598,E2 -629.9285} C_DIS
LIN {X 4.5771,Y -10.74,Z 57,A -2.9358,B 0,C 0,E1 0.1598,E2 -629.9285} C_DIS
LIN {X 5.8,Y -10.1324,Z 57,A -2.8649,B 0,C 0,E1 0.1598,E2 -629.9285} C_DIS
LIN {X 6.9063,Y -9.4133,Z 57,A -2.7935,B 0,C 0,E1 0.1598,E2 -629.9284} C_DIS
LIN {X 7.7939,Y -8.6926,Z 57,A -2.7301,B 0,C 0,E1 0.1598,E2 -629.9284} C_DIS
LIN {X 8.6606,Y -7.8295,Z 57,A -2.6612,B 0,C 0,E1 0.1598,E2 -629.9284} C_DIS
LIN {X 9.482,Y -6.8116,Z 57,A -2.5873,B 0,C 0,E1 0.1598,E2 -629.9284} C_DIS
LIN {X 10.2651,Y -5.5618,Z 57,A -2.5047,B 0,C 0,E1 0.1598,E2 -629.9286} C_DIS
LIN {X 10.6962,Y -4.6783,Z 57,A -2.4514,B 0,C 0,E1 0.1598,E2 -629.9282} C_DIS
LIN {X 11.0769,Y -3.6877,Z 57,A -2.3948,B 0,C 0,E1 0.1598,E2 -629.9282} C_DIS
LIN {X 11.343,Y -2.7638,Z 57,A -2.3454,B 0,C 0,E1 0.1598,E2 -629.9282} C_DIS
LIN {X 11.5994,Y -1.3244,Z 57,A -2.2736,B 0,C 0,E1 0.1598,E2 -629.9287} C_DIS
LIN {X 11.6745,Y -0.1433,Z 57,A -2.2205,B 0,C 0,E1 0.1598,E2 -629.9283} C_DIS
LIN {X 11.646,Y 0.8177,Z 57,A -2.1807,B 0,C 0,E1 0.1598,E2 -629.928} C_DIS
LIN {X 11.5269,Y 1.8552,Z 57,A -2.1406,B 0,C 0,E1 0.1598,E2 -629.928} C_DIS
LIN {X 11.2075,Y 3.2697,Z 57,A -2.0909,B 0,C 0,E1 0.1598,E2 -629.9287} C_DIS
LIN {X 10.7692,Y 4.508,Z 57,A -2.0545,B 0,C 0,E1 0.1598,E2 -629.9282} C_DIS
LIN {X 10.2129,Y 5.6571,Z 57,A -2.026,B 0,C 0,E1 0.1598,E2 -629.928} C_DIS
LIN {X 9.5099,Y 6.7727,Z 57,A -2.0043,B 0,C 0,E1 0.1598,E2 -629.9278} C_DIS
LIN {X 8.5389,Y 7.962,Z 57,A -1.9893,B 0,C 0,E1 0.1598,E2 -629.9279} C_DIS
LIN {X 7.6359,Y 8.8316,Z 57,A -1.9858,B 0,C 0,E1 0.1598,E2 -629.9276} C_DIS
LIN {X 6.483,Y 9.7097,Z 57,A -1.9909,B 0,C 0,E1 0.1598,E2 -629.9276} C_DIS
LIN {X 5.5925,Y 10.2484,Z 57,A -2.0012,B 0,C 0,E1 0.1598,E2 -629.9273} C_DIS
LIN {X 4.5455,Y 10.7536,Z 57,A -2.0184,B 0,C 0,E1 0.1598,E2 -629.9273} C_DIS
LIN {X 3.479,Y 11.1443,Z 57,A -2.0412,B 0,C 0,E1 0.1598,E2 -629.9273} C_DIS
LIN {X 2.1921,Y 11.4673,Z 57,A -2.0751,B 0,C 0,E1 0.1598,E2 -629.9273} C_DIS
LIN {X 0.9922,Y 11.6324,Z 57,A -2.1125,B 0,C 0,E1 0.1598,E2 -629.9273} C_DIS
LIN {X -0.0729,Y 11.6745,Z 57,A -2.1501,B 0,C 0,E1 0.1598,E2 -629.9273} C_DIS
LIN {X -1.5397,Y 11.5729,Z 57,A -2.2087,B 0,C 0,E1 0.1598,E2 -629.9273} C_DIS
LIN {X -2.892,Y 11.3108,Z 57,A -2.2697,B 0,C 0,E1 0.1598,E2 -629.9275} C_DIS
LIN {X -4.3009,Y 10.8538,Z 57,A -2.3411,B 0,C 0,E1 0.1598,E2 -629.9277} C_DIS
LIN {X -5.2852,Y 10.41,Z 57,A -2.3963,B 0,C 0,E1 0.1598,E2 -629.9277} C_DIS
LIN {X -6.8016,Y 9.489,Z 57,A -2.491,B 0,C 0,E1 0.1598,E2 -629.9282} C_DIS
LIN {X -7.9356,Y 8.5635,Z 57,A -2.5721,B 0,C 0,E1 0.1598,E2 -629.9282} C_DIS
LIN {X -8.882,Y 7.5774,Z 57,A -2.6486,B 0,C 0,E1 0.1598,E2 -629.9284} C_DIS
LIN {X -10.0228,Y 5.9876,Z 57,A -2.7571,B 0,C 0,E1 0.1598,E2 -629.9293} C_DIS
LIN {X -10.5021,Y 5.0993,Z 57,A -2.8131,B 0,C 0,E1 0.1598,E2 -629.9287} C_DIS
LIN {X -10.9225,Y 4.1227,Z 57,A -2.8699,B 0,C 0,E1 0.1598,E2 -629.9287} C_DIS
LIN {X -11.2259,Y 3.2054,Z 57,A -2.9199,B 0,C 0,E1 0.1598,E2 -629.9287} C_DIS
LIN {X -11.5204,Y 1.8942,Z 57,A -2.9857,B 0,C 0,E1 0.1598,E2 -629.9294} C_DIS
LIN {X -11.6728,Y 0.2309,Z 57,A -3.0611,B 0,C 0,E1 0.1598,E2 -629.93} C_DIS
LIN {X -11.6107,Y -1.2215,Z 57,A -3.1206,B 0,C 0,E1 0.1598,E2 -629.9296} C_DIS
LIN {X -11.317,Y -2.8676,Z 57,A -3.1789,B 0,C 0,E1 0.1598,E2 -629.9303} C_DIS
LIN {X -10.6005,Y -4.8918,Z 57,A -3.239,B 0,C 0,E1 0.1598,E2 -629.9297} C_DIS
LIN {X -9.8642,Y -6.2453,Z 57,A -3.2694,B 0,C 0,E1 0.1598,E2 -629.9297} C_DIS
LIN {X -9.2403,Y -7.136,Z 57,A -3.2848,B 0,C 0,E1 0.1598,E2 -629.9292} C_DIS
LIN {X -8.2426,Y -8.268,Z 57,A -3.2961,B 0,C 0,E1 0.1598,E2 -629.9295} C_DIS
LIN {X -7.5746,Y -8.8843,Z 57,A -3.2981,B 0,C 0,E1 0.1598,E2 -629.9292} C_DIS
LIN {X -6.7283,Y -9.5413,Z 57,A -3.2951,B 0,C 0,E1 0.1598,E2 -629.9292} C_DIS
LIN {X -5.4552,Y -10.3221,Z 57,A -3.2816,B 0,C 0,E1 0.1598,E2 -629.9292} C_DIS
LIN {X -4.4073,Y -10.8109,Z 57,A -3.2642,B 0,C 0,E1 0.1598,E2 -629.929} C_DIS
LIN {X -2.4395,Y -11.4171,Z 57,A -3.2181,B 0,C 0,E1 0.1598,E2 -629.9288} C_DIS
LIN {X -0.4685,Y -11.6653,Z 57,A -3.1567,B 0,C 0,E1 0.1598,E2 -629.9287} C_DIS
LIN {X -0.4685,Y -11.6653,Z 57,A -3.1567,B 0,C 0,E1 0.1598,E2 -629.9287} C_DIS
Enddeposition()
LIN {X 0.0353,Y -10.6863,Z 57,A -3.0949,B 0,C 0,E1 0.1598,E2 -629.9299} C_DIS
Startdeposition()
$VEL.CP = VEL_PRINT
LIN {X -1.1841,Y -10.6206,Z 57,A -3.1379,B 0,C 0,E1 0.1598,E2 -629.9287} C_DIS
LIN {X -2.1235,Y -10.4736,Z 57,A -3.1661,B 0,C 0,E1 0.1598,E2 -629.9287} C_DIS
LIN {X -3.193,Y -10.1984,Z 57,A -3.1935,B 0,C 0,E1 0.1598,E2 -629.9287} C_DIS
LIN {X -4.2966,Y -9.7826,Z 57,A -3.2161,B 0,C 0,E1 0.1598,E2 -629.9288} C_DIS
LIN {X -5.1157,Y -9.3828,Z 57,A -3.2291,B 0,C 0,E1 0.1598,E2 -629.9288} C_DIS
LIN {X -6.0125,Y -8.835,Z 57,A -3.2386,B 0,C 0,E1 0.1598,E2 -629.9289} C_DIS
LIN {X -6.7462,Y -8.2882,Z 57,A -3.2422,B 0,C 0,E1 0.1598,E2 -629.9289} C_DIS
LIN {X -7.9271,Y -7.1671,Z 57,A -3.2373,B 0,C 0,E1 0.1598,E2 -629.9294} C_DIS
LIN {X -9.0933,Y -5.6136,Z 57,A -3.2142,B 0,C 0,E1 0.1598,E2 -629.9294} C_DIS
LIN {X -9.8207,Y -4.2133,Z 57,A -3.1811,B 0,C 0,E1 0.1598,E2 -629.9297} C_DIS
LIN {X -10.197,Y -3.1966,Z 57,A -3.1523,B 0,C 0,E1 0.1598,E2 -629.9292} C_DIS
LIN {X -10.4874,Y -2.0545,Z 57,A -3.1144,B 0,C 0,E1 0.1598,E2 -629.9292} C_DIS
LIN {X -10.6431,Y -0.9635,Z 57,A -3.0739,B 0,C 0,E1 0.1598,E2 -629.9292} C_DIS
LIN {X -10.6884,Y 0.0212,Z 57,A -3.0341,B 0,C 0,E1 0.1598,E2 -629.9289} C_DIS
LIN {X -10.6095,Y 1.2799,Z 57,A -2.9776,B 0,C 0,E1 0.1598,E2 -629.9292} C_DIS
LIN {X -10.3951,Y 2.4633,Z 57,A -2.9197,B 0,C 0,E1 0.1598,E2 -629.929} C_DIS
LIN {X -10.1981,Y 3.1822,Z 57,A -2.8825,B 0,C 0,E1 0.1598,E2 -629.9286} C_DIS
LIN {X -9.9515,Y 3.8857,Z 57,A -2.8437,B 0,C 0,E1 0.1598,E2 -629.9285} C_DIS
LIN {X -9.5778,Y 4.7393,Z 57,A -2.7936,B 0,C 0,E1 0.1598,E2 -629.9285} C_DIS
LIN {X -8.9698,Y 5.8095,Z 57,A -2.7257,B 0,C 0,E1 0.1598,E2 -629.9287} C_DIS
LIN {X -8.1056,Y 6.9647,Z 57,A -2.6448,B 0,C 0,E1 0.1598,E2 -629.9287} C_DIS
LIN {X -6.9284,Y 8.1365,Z 57,A -2.5518,B 0,C 0,E1 0.1598,E2 -629.9285} C_DIS
LIN {X -5.3599,Y 9.2452,Z 57,A -2.4473,B 0,C 0,E1 0.1598,E2 -629.928} C_DIS
LIN {X -4.5565,Y 9.6665,Z 57,A -2.4,B 0,C 0,E1 0.1598,E2 -629.9278} C_DIS
LIN {X -3.4308,Y 10.1209,Z 57,A -2.3392,B 0,C 0,E1 0.1598,E2 -629.9277} C_DIS
LIN {X -2.1136,Y 10.4756,Z 57,A -2.2755,B 0,C 0,E1 0.1598,E2 -629.9275} C_DIS
LIN {X -0.3805,Y 10.6796,Z 57,A -2.2028,B 0,C 0,E1 0.1598,E2 -629.9274} C_DIS
LIN {X 0.8533,Y 10.6524,Z 57,A -2.1584,B 0,C 0,E1 0.1598,E2 -629.9274} C_DIS
LIN {X 2.1161,Y 10.4751,Z 57,A -2.1192,B 0,C 0,E1 0.1598,E2 -629.9273} C_DIS
LIN {X 3.3345,Y 10.1527,Z 57,A -2.0879,B 0,C 0,E1 0.1598,E2 -629.9273} C_DIS
LIN {X 4.6229,Y 9.6344,Z 57,A -2.0622,B 0,C 0,E1 0.1598,E2 -629.9273} C_DIS
LIN {X 5.8208,Y 8.9625,Z 57,A -2.0465,B 0,C 0,E1 0.1598,E2 -629.9275} C_DIS
LIN {X 6.8977,Y 8.1597,Z 57,A -2.0409,B 0,C 0,E1 0.1598,E2 -629.9275} C_DIS
LIN {X 7.5879,Y 7.5252,Z 57,A -2.0425,B 0,C 0,E1 0.1598,E2 -629.9275} C_DIS
LIN {X 8.4017,Y 6.6045,Z 57,A -2.0516,B 0,C 0,E1 0.1598,E2 -629.9278} C_DIS
LIN {X 9.0974,Y 5.6076,Z 57,A -2.0685,B 0,C 0,E1 0.1598,E2 -629.9278} C_DIS
LIN {X 9.6918,Y 4.5024,Z 57,A -2.0937,B 0,C 0,E1 0.1598,E2 -629.928} C_DIS
LIN {X 10.1071,Y 3.4709,Z 57,A -2.1221,B 0,C 0,E1 0.1598,E2 -629.9284} C_DIS
LIN {X 10.5924,Y 1.4167,Z 57,A -2.1908,B 0,C 0,E1 0.1598,E2 -629.9298} C_DIS
LIN {X 10.5924,Y 1.4167,Z 57,A -2.192,B 0,C 0,E1 0.1598,E2 -629.9286} C_DIS
LIN {X 10.6856,Y -0.1683,Z 57,A -2.2563,B 0,C 0,E1 0.1598,E2 -629.9289} C_DIS
LIN {X 10.628,Y -1.0936,Z 57,A -2.2989,B 0,C 0,E1 0.1598,E2 -629.928} C_DIS
LIN {X 10.4957,Y -2.0113,Z 57,A -2.3431,B 0,C 0,E1 0.1598,E2 -629.9281} C_DIS
LIN {X 10.233,Y -3.08,Z 57,A -2.3985,B 0,C 0,E1 0.1598,E2 -629.9282} C_DIS
LIN {X 9.7884,Y -4.2884,Z 57,A -2.4664,B 0,C 0,E1 0.1598,E2 -629.9285} C_DIS
LIN {X 9.2355,Y -5.3774,Z 57,A -2.5335,B 0,C 0,E1 0.1598,E2 -629.9285} C_DIS
LIN {X 8.0956,Y -6.9764,Z 57,A -2.6431,B 0,C 0,E1 0.1598,E2 -629.9293} C_DIS
LIN {X 7.1127,Y -7.9761,Z 57,A -2.7228,B 0,C 0,E1 0.1598,E2 -629.9285} C_DIS
LIN {X 5.9792,Y -8.8573,Z 57,A -2.8021,B 0,C 0,E1 0.1598,E2 -629.9285} C_DIS
LIN {X 5.0598,Y -9.4129,Z 57,A -2.8598,B 0,C 0,E1 0.1598,E2 -629.9284} C_DIS
LIN {X 3.5416,Y -10.0823,Z 57,A -2.944,B 0,C 0,E1 0.1598,E2 -629.9286} C_DIS
LIN {X 2.2546,Y -10.446,Z 57,A -3.0068,B 0,C 0,E1 0.1598,E2 -629.9285} C_DIS
LIN {X 0.4712,Y -10.6762,Z 57,A -3.0819,B 0,C 0,E1 0.1598,E2 -629.9285} C_DIS
LIN {X 0.4712,Y -10.6762,Z 57,A -3.0819,B 0,C 0,E1 0.1598,E2 -629.9285} C_DIS
Enddeposition()
LIN {X 0.0216,Y -9.6977,Z 57,A -3.055,B 0,C 0,E1 0.1598,E2 -629.9299} C_DIS
Startdeposition()
$VEL.CP = VEL_PRINT
LIN {X 0.9982,Y -9.6469,Z 57,A -3.0183,B 0,C 0,E1 0.1598,E2 -629.9285} C_DIS
LIN {X 2.2879,Y -9.4246,Z 57,A -2.9617,B 0,C 0,E1 0.1598,E2 -629.9284} C_DIS
LIN {X 3.7982,Y -8.9231,Z 57,A -2.8848,B 0,C 0,E1 0.1598,E2 -629.9284} C_DIS
LIN {X 5.3376,Y -8.0974,Z 57,A -2.793,B 0,C 0,E1 0.1598,E2 -629.9284} C_DIS
LIN {X 6.5797,Y -7.1214,Z 57,A -2.7055,B 0,C 0,E1 0.1598,E2 -629.9284} C_DIS
LIN {X 7.2874,Y -6.3996,Z 57,A -2.6486,B 0,C 0,E1 0.1598,E2 -629.9284} C_DIS
LIN {X 8.1197,Y -5.2984,Z 57,A -2.5708,B 0,C 0,E1 0.1598,E2 -629.9284} C_DIS
LIN {X 8.5133,Y -4.6387,Z 57,A -2.5284,B 0,C 0,E1 0.1598,E2 -629.9281} C_DIS
LIN {X 8.9883,Y -3.6422,Z 57,A -2.468,B 0,C 0,E1 0.1598,E2 -629.9282} C_DIS
LIN {X 9.3384,Y -2.6173,Z 57,A -2.4111,B 0,C 0,E1 0.1598,E2 -629.9283} C_DIS
LIN {X 9.5966,Y -1.4031,Z 57,A -2.3494,B 0,C 0,E1 0.1598,E2 -629.9284} C_DIS
LIN {X 9.694,Y -0.2909,Z 57,A -2.2983,B 0,C 0,E1 0.1598,E2 -629.9282} C_DIS
LIN {X 9.6271,Y 1.1727,Z 57,A -2.2377,B 0,C 0,E1 0.1598,E2 -629.9286} C_DIS
LIN {X 9.4493,Y 2.1836,Z 57,A -2.2015,B 0,C 0,E1 0.1598,E2 -629.928} C_DIS
LIN {X 9.1245,Y 3.2767,Z 57,A -2.1666,B 0,C 0,E1 0.1598,E2 -629.928} C_DIS
LIN {X 8.6821,Y 4.3219,Z 57,A -2.1383,B 0,C 0,E1 0.1598,E2 -629.928} C_DIS
LIN {X 8.1972,Y 5.1832,Z 57,A -2.1196,B 0,C 0,E1 0.1598,E2 -629.9277} C_DIS
LIN {X 7.6309,Y 5.9861,Z 57,A -2.1062,B 0,C 0,E1 0.1598,E2 -629.9277} C_DIS
LIN {X 6.7556,Y 6.9588,Z 57,A -2.0967,B 0,C 0,E1 0.1598,E2 -629.9278} C_DIS
LIN {X 5.9039,Y 7.6945,Z 57,A -2.097,B 0,C 0,E1 0.1598,E2 -629.9276} C_DIS
LIN {X 4.8717,Y 8.386,Z 57,A -2.1057,B 0,C 0,E1 0.1598,E2 -629.9276} C_DIS
LIN {X 3.7881,Y 8.9278,Z 57,A -2.1227,B 0,C 0,E1 0.1598,E2 -629.9275} C_DIS
LIN {X 2.6275,Y 9.332,Z 57,A -2.1485,B 0,C 0,E1 0.1598,E2 -629.9275} C_DIS
LIN {X 1.5511,Y 9.5739,Z 57,A -2.178,B 0,C 0,E1 0.1598,E2 -629.9274} C_DIS
LIN {X 0.5807,Y 9.6808,Z 57,A -2.2094,B 0,C 0,E1 0.1598,E2 -629.9274} C_DIS
LIN {X -0.6879,Y 9.6738,Z 57,A -2.2565,B 0,C 0,E1 0.1598,E2 -629.9274} C_DIS
LIN {X -1.697,Y 9.549,Z 57,A -2.2991,B 0,C 0,E1 0.1598,E2 -629.9275} C_DIS
LIN {X -2.9395,Y 9.242,Z 57,A -2.358,B 0,C 0,E1 0.1598,E2 -629.9276} C_DIS
LIN {X -4.3413,Y 8.6724,Z 57,A -2.4338,B 0,C 0,E1 0.1598,E2 -629.9278} C_DIS
LIN {X -5.4509,Y 8.0184,Z 57,A -2.5024,B 0,C 0,E1 0.1598,E2 -629.928} C_DIS
LIN {X -6.2929,Y 7.3799,Z 57,A -2.5605,B 0,C 0,E1 0.1598,E2 -629.928} C_DIS
LIN {X -7.1428,Y 6.5602,Z 57,A -2.6265,B 0,C 0,E1 0.1598,E2 -629.9283} C_DIS
LIN {X -7.8984,Y 5.6283,Z 57,A -2.6937,B 0,C 0,E1 0.1598,E2 -629.9285} C_DIS
LIN {X -8.4058,Y 4.8374,Z 57,A -2.746,B 0,C 0,E1 0.1598,E2 -629.9284} C_DIS
LIN {X -8.9314,Y 3.7799,Z 57,A -2.8099,B 0,C 0,E1 0.1598,E2 -629.9287} C_DIS
LIN {X -9.3691,Y 2.5035,Z 57,A -2.8797,B 0,C 0,E1 0.1598,E2 -629.9291} C_DIS
LIN {X -9.6511,Y 0.9546,Z 57,A -2.9552,B 0,C 0,E1 0.1598,E2 -629.9297} C_DIS
LIN {X -9.6974,Y -0.1558,Z 57,A -3.0046,B 0,C 0,E1 0.1598,E2 -629.9291} C_DIS
LIN {X -9.4783,Y -2.0533,Z 57,A -3.0758,B 0,C 0,E1 0.1598,E2 -629.9303} C_DIS
LIN {X -9.2356,Y -2.9594,Z 57,A -3.1062,B 0,C 0,E1 0.1598,E2 -629.9294} C_DIS
LIN {X -8.6992,Y -4.2873,Z 57,A -3.1428,B 0,C 0,E1 0.1598,E2 -629.9294} C_DIS
LIN {X -7.821,Y -5.7353,Z 57,A -3.1718,B 0,C 0,E1 0.1598,E2 -629.9297} C_DIS
LIN {X -7.1141,Y -6.5918,Z 57,A -3.1828,B 0,C 0,E1 0.1598,E2 -629.9292} C_DIS
LIN {X -6.2902,Y -7.3822,Z 57,A -3.1863,B 0,C 0,E1 0.1598,E2 -629.929} C_DIS
LIN {X -5.6387,Y -7.8908,Z 57,A -3.1842,B 0,C 0,E1 0.1598,E2 -629.9289} C_DIS
LIN {X -4.7755,Y -8.4414,Z 57,A -3.176,B 0,C 0,E1 0.1598,E2 -629.9289} C_DIS
LIN {X -3.678,Y -8.9736,Z 57,A -3.1585,B 0,C 0,E1 0.1598,E2 -629.9289} C_DIS
LIN {X -1.8084,Y -9.5284,Z 57,A -3.1136,B 0,C 0,E1 0.1598,E2 -629.9288} C_DIS
LIN {X -0.2679,Y -9.6935,Z 57,A -3.0644,B 0,C 0,E1 0.1598,E2 -629.9285} C_DIS
LIN {X -0.2679,Y -9.6935,Z 57,A -3.0644,B 0,C 0,E1 0.1598,E2 -629.9285} C_DIS
Enddeposition()
LIN {X -0.0044,Y -8.7092,Z 57,A -3.0112,B 0,C 0,E1 0.1598,E2 -629.9298} C_DIS
Startdeposition()
$VEL.CP = VEL_PRINT
LIN {X -0.8894,Y -8.6643,Z 57,A -3.043,B 0,C 0,E1 0.1598,E2 -629.9286} C_DIS
LIN {X -2.0014,Y -8.477,Z 57,A -3.0758,B 0,C 0,E1 0.1598,E2 -629.9286} C_DIS
LIN {X -2.9051,Y -8.2112,Z 57,A -3.0975,B 0,C 0,E1 0.1598,E2 -629.9286} C_DIS
LIN {X -4.2271,Y -7.6157,Z 57,A -3.1204,B 0,C 0,E1 0.1598,E2 -629.9288} C_DIS
LIN {X -5.1532,Y -7.0223,Z 57,A -3.1292,B 0,C 0,E1 0.1598,E2 -629.9288} C_DIS
LIN {X -5.971,Y -6.3416,Z 57,A -3.1301,B 0,C 0,E1 0.1598,E2 -629.9288} C_DIS
LIN {X -6.7144,Y -5.5486,Z 57,A -3.1236,B 0,C 0,E1 0.1598,E2 -629.929} C_DIS
LIN {X -7.363,Y -4.653,Z 57,A -3.1093,B 0,C 0,E1 0.1598,E2 -629.929} C_DIS
LIN {X -7.9923,Y -3.4624,Z 57,A -3.0816,B 0,C 0,E1 0.1598,E2 -629.9292} C_DIS
LIN {X -8.3276,Y -2.5389,Z 57,A -3.055,B 0,C 0,E1 0.1598,E2 -629.9289} C_DIS
LIN {X -8.5645,Y -1.5855,Z 57,A -3.0232,B 0,C 0,E1 0.1598,E2 -629.929} C_DIS
LIN {X -8.709,Y -0.1555,Z 57,A -2.9674,B 0,C 0,E1 0.1598,E2 -629.9294} C_DIS
LIN {X -8.6528,Y 0.9983,Z 57,A -2.9166,B 0,C 0,E1 0.1598,E2 -629.9291} C_DIS
LIN {X -8.2951,Y 2.6562,Z 57,A -2.8324,B 0,C 0,E1 0.1598,E2 -629.9299} C_DIS
LIN {X -7.7512,Y 3.9726,Z 57,A -2.7574,B 0,C 0,E1 0.1598,E2 -629.929} C_DIS
LIN {X -7.2384,Y 4.8452,Z 57,A -2.7018,B 0,C 0,E1 0.1598,E2 -629.9286} C_DIS
LIN {X -6.5185,Y 5.7775,Z 57,A -2.6359,B 0,C 0,E1 0.1598,E2 -629.9284} C_DIS
LIN {X -5.7409,Y 6.5465,Z 57,A -2.5747,B 0,C 0,E1 0.1598,E2 -629.9282} C_DIS
LIN {X -4.8516,Y 7.2341,Z 57,A -2.5128,B 0,C 0,E1 0.1598,E2 -629.928} C_DIS
LIN {X -4.1383,Y 7.6639,Z 57,A -2.4684,B 0,C 0,E1 0.1598,E2 -629.9278} C_DIS
LIN {X -3.0987,Y 8.1402,Z 57,A -2.4098,B 0,C 0,E1 0.1598,E2 -629.9278} C_DIS
LIN {X -1.9169,Y 8.4965,Z 57,A -2.3511,B 0,C 0,E1 0.1598,E2 -629.9276} C_DIS
LIN {X -0.7343,Y 8.679,Z 57,A -2.2998,B 0,C 0,E1 0.1598,E2 -629.9276} C_DIS
LIN {X 0.7705,Y 8.6757,Z 57,A -2.2443,B 0,C 0,E1 0.1598,E2 -629.9274} C_DIS
LIN {X 1.702,Y 8.5422,Z 57,A -2.2156,B 0,C 0,E1 0.1598,E2 -629.9274} C_DIS
LIN {X 3.4045,Y 8.0172,Z 57,A -2.1749,B 0,C 0,E1 0.1598,E2 -629.9275} C_DIS
LIN {X 4.027,Y 7.7229,Z 57,A -2.1646,B 0,C 0,E1 0.1598,E2 -629.9275} C_DIS
LIN {X 4.9053,Y 7.1978,Z 57,A -2.1544,B 0,C 0,E1 0.1598,E2 -629.9275} C_DIS
LIN {X 5.6277,Y 6.6481,Z 57,A -2.1512,B 0,C 0,E1 0.1598,E2 -629.9275} C_DIS
LIN {X 6.3241,Y 5.9896,Z 57,A -2.1536,B 0,C 0,E1 0.1598,E2 -629.9275} C_DIS
LIN {X 6.9549,Y 5.2439,Z 57,A -2.1621,B 0,C 0,E1 0.1598,E2 -629.9276} C_DIS
LIN {X 7.596,Y 4.2565,Z 57,A -2.1803,B 0,C 0,E1 0.1598,E2 -629.928} C_DIS
LIN {X 7.9624,Y 3.5306,Z 57,A -2.1979,B 0,C 0,E1 0.1598,E2 -629.9279} C_DIS
LIN {X 8.5183,Y 1.8181,Z 57,A -2.2502,B 0,C 0,E1 0.1598,E2 -629.9284} C_DIS
LIN {X 8.7101,Y -0.0976,Z 57,A -2.3241,B 0,C 0,E1 0.1598,E2 -629.9295} C_DIS
LIN {X 8.5848,Y -1.4739,Z 57,A -2.3885,B 0,C 0,E1 0.1598,E2 -629.9287} C_DIS
LIN {X 8.3077,Y -2.6054,Z 57,A -2.4474,B 0,C 0,E1 0.1598,E2 -629.9284} C_DIS
LIN {X 7.9213,Y -3.6221,Z 57,A -2.5053,B 0,C 0,E1 0.1598,E2 -629.9284} C_DIS
LIN {X 7.4526,Y -4.5024,Z 57,A -2.5603,B 0,C 0,E1 0.1598,E2 -629.9282} C_DIS
LIN {X 6.5483,Y -5.7435,Z 57,A -2.6461,B 0,C 0,E1 0.1598,E2 -629.9289} C_DIS
LIN {X 5.501,Y -6.7533,Z 57,A -2.7281,B 0,C 0,E1 0.1598,E2 -629.9286} C_DIS
LIN {X 4.0301,Y -7.7218,Z 57,A -2.8235,B 0,C 0,E1 0.1598,E2 -629.9286} C_DIS
LIN {X 2.6553,Y -8.2951,Z 57,A -2.8987,B 0,C 0,E1 0.1598,E2 -629.9285} C_DIS
LIN {X 1.4578,Y -8.5875,Z 57,A -2.9551,B 0,C 0,E1 0.1598,E2 -629.9285} C_DIS
LIN {X -0.0044,Y -8.7092,Z 57,A -3.0139,B 0,C 0,E1 0.1598,E2 -629.9285} C_DIS
Enddeposition()
LIN {X -0.0044,Y -8.7092,Z 57,A -3.0139,B 0,C 0,E1 0.1598,E2 -629.9285} C_DIS
Startdeposition()
$VEL.CP = VEL_PRINT
LIN {X 0.0659,Y -7.7219,Z 57,A -2.9684,B 0,C 0,E1 0.1598,E2 -629.929} C_DIS
LIN {X 1.9365,Y -7.4751,Z 57,A -2.8898,B 0,C 0,E1 0.1598,E2 -629.9283} C_DIS
LIN {X 3.284,Y -6.9887,Z 57,A -2.8196,B 0,C 0,E1 0.1598,E2 -629.9283} C_DIS
LIN {X 4.0007,Y -6.6048,Z 57,A -2.7769,B 0,C 0,E1 0.1598,E2 -629.9283} C_DIS
LIN {X 4.9515,Y -5.9256,Z 57,A -2.7129,B 0,C 0,E1 0.1598,E2 -629.9283} C_DIS
LIN {X 6.0329,Y -4.8202,Z 57,A -2.6256,B 0,C 0,E1 0.1598,E2 -629.9285} C_DIS
LIN {X 6.9428,Y -3.3792,Z 57,A -2.53,B 0,C 0,E1 0.1598,E2 -629.9289} C_DIS
LIN {X 7.4288,Y -2.107,Z 57,A -2.458,B 0,C 0,E1 0.1598,E2 -629.9286} C_DIS
LIN {X 7.6678,Y -0.9133,Z 57,A -2.3982,B 0,C 0,E1 0.1598,E2 -629.9284} C_DIS
LIN {X 7.7103,Y 0.4204,Z 57,A -2.3394,B 0,C 0,E1 0.1598,E2 -629.9285} C_DIS
LIN {X 7.5748,Y 1.5011,Z 57,A -2.2984,B 0,C 0,E1 0.1598,E2 -629.9282} C_DIS
LIN {X 7.287,Y 2.5542,Z 57,A -2.264,B 0,C 0,E1 0.1598,E2 -629.9282} C_DIS
LIN {X 6.8367,Y 3.5901,Z 57,A -2.2364,B 0,C 0,E1 0.1598,E2 -629.928} C_DIS
LIN {X 6.2957,Y 4.4716,Z 57,A -2.2189,B 0,C 0,E1 0.1598,E2 -629.9279} C_DIS
LIN {X 5.6158,Y 5.3003,Z 57,A -2.2086,B 0,C 0,E1 0.1598,E2 -629.9278} C_DIS
LIN {X 4.8441,Y 6.0138,Z 57,A -2.2067,B 0,C 0,E1 0.1598,E2 -629.9277} C_DIS
LIN {X 3.954,Y 6.633,Z 57,A -2.2132,B 0,C 0,E1 0.1598,E2 -629.9277} C_DIS
LIN {X 2.889,Y 7.1609,Z 57,A -2.2301,B 0,C 0,E1 0.1598,E2 -629.9276} C_DIS
LIN {X 1.4464,Y 7.5853,Z 57,A -2.2653,B 0,C 0,E1 0.1598,E2 -629.9276} C_DIS
LIN {X 0.1102,Y 7.7211,Z 57,A -2.309,B 0,C 0,E1 0.1598,E2 -629.9276} C_DIS
LIN {X -1.0565,Y 7.6489,Z 57,A -2.3551,B 0,C 0,E1 0.1598,E2 -629.9276} C_DIS
LIN {X -2.3676,Y 7.3499,Z 57,A -2.4162,B 0,C 0,E1 0.1598,E2 -629.9276} C_DIS
LIN {X -3.3678,Y 6.9488,Z 57,A -2.4701,B 0,C 0,E1 0.1598,E2 -629.9278} C_DIS
LIN {X -4.3622,Y 6.3719,Z 57,A -2.5311,B 0,C 0,E1 0.1598,E2 -629.928} C_DIS
LIN {X -5.631,Y 5.284,Z 57,A -2.6236,B 0,C 0,E1 0.1598,E2 -629.9286} C_DIS
LIN {X -6.5439,Y 4.0996,Z 57,A -2.7073,B 0,C 0,E1 0.1598,E2 -629.9288} C_DIS
LIN {X -7.1336,Y 2.9561,Z 57,A -2.7776,B 0,C 0,E1 0.1598,E2 -629.9288} C_DIS
LIN {X -7.5548,Y 1.5979,Z 57,A -2.8503,B 0,C 0,E1 0.1598,E2 -629.9293} C_DIS
LIN {X -7.6997,Y 0.5837,Z 57,A -2.899,B 0,C 0,E1 0.1598,E2 -629.9289} C_DIS
LIN {X -7.7087,Y -0.4481,Z 57,A -2.9431,B 0,C 0,E1 0.1598,E2 -629.9289} C_DIS
LIN {X -7.5784,Y -1.4827,Z 57,A -2.9819,B 0,C 0,E1 0.1598,E2 -629.9293} C_DIS
LIN {X -7.2305,Y -2.7103,Z 57,A -3.0213,B 0,C 0,E1 0.1598,E2 -629.9292} C_DIS
LIN {X -6.3931,Y -4.331,Z 57,A -3.0594,B 0,C 0,E1 0.1598,E2 -629.9292} C_DIS
LIN {X -5.8039,Y -5.0937,Z 57,A -3.0706,B 0,C 0,E1 0.1598,E2 -629.9288} C_DIS
LIN {X -4.959,Y -5.9131,Z 57,A -3.0743,B 0,C 0,E1 0.1598,E2 -629.9289} C_DIS
LIN {X -4.2727,Y -6.4279,Z 57,A -3.0713,B 0,C 0,E1 0.1598,E2 -629.9287} C_DIS
LIN {X -3.0322,Y -7.1012,Z 57,A -3.0543,B 0,C 0,E1 0.1598,E2 -629.9287} C_DIS
LIN {X -1.1547,Y -7.6353,Z 57,A -3.0084,B 0,C 0,E1 0.1598,E2 -629.9287} C_DIS
LIN {X 0.0014,Y -7.7215,Z 57,A -2.9698,B 0,C 0,E1 0.1598,E2 -629.9284} C_DIS
Enddeposition()
LIN {X 0.0014,Y -7.7215,Z 57,A -2.9698,B 0,C 0,E1 0.1598,E2 -629.9284} C_DIS
Startdeposition()
$VEL.CP = VEL_PRINT
LIN {X -0.26,Y -6.7285,Z 57,A -2.9362,B 0,C 0,E1 0.1598,E2 -629.929} C_DIS
LIN {X -1.307,Y -6.6022,Z 57,A -2.9698,B 0,C 0,E1 0.1598,E2 -629.9284} C_DIS
LIN {X -2.0071,Y -6.423,Z 57,A -2.9879,B 0,C 0,E1 0.1598,E2 -629.9284} C_DIS
LIN {X -2.6841,Y -6.1703,Z 57,A -3.0019,B 0,C 0,E1 0.1598,E2 -629.9284} C_DIS
LIN {X -3.3309,Y -5.8481,Z 57,A -3.0119,B 0,C 0,E1 0.1598,E2 -629.9285} C_DIS
LIN {X -4.0862,Y -5.3524,Z 57,A -3.0184,B 0,C 0,E1 0.1598,E2 -629.9286} C_DIS
LIN {X -4.8152,Y -4.7073,Z 57,A -3.0177,B 0,C 0,E1 0.1598,E2 -629.9286} C_DIS
LIN {X -5.5563,Y -3.7979,Z 57,A -3.0059,B 0,C 0,E1 0.1598,E2 -629.9289} C_DIS
LIN {X -6.0677,Y -2.9197,Z 57,A -2.9872,B 0,C 0,E1 0.1598,E2 -629.9291} C_DIS
LIN {X -6.4485,Y -1.9382,Z 57,A -2.9597,B 0,C 0,E1 0.1598,E2 -629.9289} C_DIS
LIN {X -6.7246,Y -0.3463,Z 57,A -2.9014,B 0,C 0,E1 0.1598,E2 -629.9297} C_DIS
LIN {X -6.7057,Y 0.6131,Z 57,A -2.8608,B 0,C 0,E1 0.1598,E2 -629.9288} C_DIS
LIN {X -6.5603,Y 1.518,Z 57,A -2.8173,B 0,C 0,E1 0.1598,E2 -629.9286} C_DIS
LIN {X -6.2902,Y 2.4027,Z 57,A -2.7698,B 0,C 0,E1 0.1598,E2 -629.9286} C_DIS
LIN {X -5.8305,Y 3.3688,Z 57,A -2.7118,B 0,C 0,E1 0.1598,E2 -629.9286} C_DIS
LIN {X -5.3474,Y 4.0925,Z 57,A -2.6635,B 0,C 0,E1 0.1598,E2 -629.9283} C_DIS
LIN {X -4.6118,Y 4.898,Z 57,A -2.6022,B 0,C 0,E1 0.1598,E2 -629.9283} C_DIS
LIN {X -3.9395,Y 5.4544,Z 57,A -2.5539,B 0,C 0,E1 0.1598,E2 -629.928} C_DIS
LIN {X -2.9502,Y 6.053,Z 57,A -2.4921,B 0,C 0,E1 0.1598,E2 -629.928} C_DIS
LIN {X -2.0166,Y 6.4244,Z 57,A -2.4419,B 0,C 0,E1 0.1598,E2 -629.9278} C_DIS
LIN {X -1.3069,Y 6.6011,Z 57,A -2.4083,B 0,C 0,E1 0.1598,E2 -629.9277} C_DIS
LIN {X -0.5711,Y 6.7093,Z 57,A -2.3766,B 0,C 0,E1 0.1598,E2 -629.9277} C_DIS
LIN {X 0.9141,Y 6.6715,Z 57,A -2.3234,B 0,C 0,E1 0.1598,E2 -629.9275} C_DIS
LIN {X 2.3024,Y 6.3202,Z 57,A -2.287,B 0,C 0,E1 0.1598,E2 -629.9275} C_DIS
LIN {X 3.2661,Y 5.8887,Z 57,A -2.2698,B 0,C 0,E1 0.1598,E2 -629.9276} C_DIS
LIN {X 4.1187,Y 5.3274,Z 57,A -2.2622,B 0,C 0,E1 0.1598,E2 -629.9276} C_DIS
LIN {X 4.8546,Y 4.6666,Z 57,A -2.2632,B 0,C 0,E1 0.1598,E2 -629.9277} C_DIS
LIN {X 5.5204,Y 3.8492,Z 57,A -2.2734,B 0,C 0,E1 0.1598,E2 -629.9279} C_DIS
LIN {X 6.0633,Y 2.9289,Z 57,A -2.2926,B 0,C 0,E1 0.1598,E2 -629.928} C_DIS
LIN {X 6.5281,Y 1.6482,Z 57,A -2.3298,B 0,C 0,E1 0.1598,E2 -629.9284} C_DIS
LIN {X 6.713,Y 0.5217,Z 57,A -2.3713,B 0,C 0,E1 0.1598,E2 -629.9284} C_DIS
LIN {X 6.6687,Y -0.9346,Z 57,A -2.4346,B 0,C 0,E1 0.1598,E2 -629.929} C_DIS
LIN {X 6.3891,Y -2.1237,Z 57,A -2.4958,B 0,C 0,E1 0.1598,E2 -629.929} C_DIS
LIN {X 5.8297,Y -3.3694,Z 57,A -2.57,B 0,C 0,E1 0.1598,E2 -629.9287} C_DIS
LIN {X 5.0314,Y -4.4696,Z 57,A -2.6465,B 0,C 0,E1 0.1598,E2 -629.9286} C_DIS
LIN {X 4.3038,Y -5.1789,Z 57,A -2.7037,B 0,C 0,E1 0.1598,E2 -629.9285} C_DIS
LIN {X 3.2399,Y -5.9031,Z 57,A -2.7738,B 0,C 0,E1 0.1598,E2 -629.9284} C_DIS
LIN {X 2.3904,Y -6.2903,Z 57,A -2.8217,B 0,C 0,E1 0.1598,E2 -629.9283} C_DIS
LIN {X 1.6787,Y -6.5171,Z 57,A -2.8575,B 0,C 0,E1 0.1598,E2 -629.9283} C_DIS
LIN {X 0.946,Y -6.6611,Z 57,A -2.8906,B 0,C 0,E1 0.1598,E2 -629.9283} C_DIS
LIN {X 0.0153,Y -6.7324,Z 57,A -2.9277,B 0,C 0,E1 0.1598,E2 -629.9283} C_DIS
Enddeposition()
LIN {X 0.0153,Y -6.7324,Z 57,A -2.9277,B 0,C 0,E1 0.1598,E2 -629.9283} C_DIS
Startdeposition()
$VEL.CP = VEL_PRINT
LIN {X 0.5847,Y -5.7107,Z 57,A -2.8624,B 0,C 0,E1 0.1598,E2 -629.9289} C_DIS
LIN {X 1.3786,Y -5.5718,Z 57,A -2.828,B 0,C 0,E1 0.1598,E2 -629.9282} C_DIS
LIN {X 2.4697,Y -5.1874,Z 57,A -2.7715,B 0,C 0,E1 0.1598,E2 -629.9282} C_DIS
LIN {X 3.2399,Y -4.7388,Z 57,A -2.7241,B 0,C 0,E1 0.1598,E2 -629.9282} C_DIS
LIN {X 4.1036,Y -4.0211,Z 57,A -2.6615,B 0,C 0,E1 0.1598,E2 -629.9282} C_DIS
LIN {X 4.5711,Y -3.4744,Z 57,A -2.6211,B 0,C 0,E1 0.1598,E2 -629.9281} C_DIS
LIN {X 5.0197,Y -2.7814,Z 57,A -2.5749,B 0,C 0,E1 0.1598,E2 -629.9281} C_DIS
LIN {X 5.367,Y -2.0328,Z 57,A -2.5301,B 0,C 0,E1 0.1598,E2 -629.9281} C_DIS
LIN {X 5.666,Y -0.9536,Z 57,A -2.4728,B 0,C 0,E1 0.1598,E2 -629.9283} C_DIS
LIN {X 5.7453,Y 0.0075,Z 57,A -2.4287,B 0,C 0,E1 0.1598,E2 -629.9283} C_DIS
LIN {X 5.698,Y 0.6956,Z 57,A -2.4013,B 0,C 0,E1 0.1598,E2 -629.928} C_DIS
LIN {X 5.5539,Y 1.4706,Z 57,A -2.3734,B 0,C 0,E1 0.1598,E2 -629.928} C_DIS
LIN {X 5.2406,Y 2.3428,Z 57,A -2.3478,B 0,C 0,E1 0.1598,E2 -629.928} C_DIS
LIN {X 4.8947,Y 2.9985,Z 57,A -2.3327,B 0,C 0,E1 0.1598,E2 -629.9278} C_DIS
LIN {X 4.4661,Y 3.6034,Z 57,A -2.3227,B 0,C 0,E1 0.1598,E2 -629.9278} C_DIS
LIN {X 3.9666,Y 4.1512,Z 57,A -2.3178,B 0,C 0,E1 0.1598,E2 -629.9278} C_DIS
LIN {X 3.3979,Y 4.6269,Z 57,A -2.3185,B 0,C 0,E1 0.1598,E2 -629.9277} C_DIS
LIN {X 2.7735,Y 5.0267,Z 57,A -2.3245,B 0,C 0,E1 0.1598,E2 -629.9277} C_DIS
LIN {X 2.1016,Y 5.3398,Z 57,A -2.336,B 0,C 0,E1 0.1598,E2 -629.9277} C_DIS
LIN {X 1.2167,Y 5.6151,Z 57,A -2.3569,B 0,C 0,E1 0.1598,E2 -629.9277} C_DIS
LIN {X -0.1677,Y 5.743,Z 57,A -2.4026,B 0,C 0,E1 0.1598,E2 -629.9277} C_DIS
LIN {X -1.1649,Y 5.6262,Z 57,A -2.4443,B 0,C 0,E1 0.1598,E2 -629.9277} C_DIS
LIN {X -2.2723,Y 5.2711,Z 57,A -2.5002,B 0,C 0,E1 0.1598,E2 -629.9278} C_DIS
LIN {X -3.0115,Y 4.8871,Z 57,A -2.5437,B 0,C 0,E1 0.1598,E2 -629.9278} C_DIS
LIN {X -3.8479,Y 4.2668,Z 57,A -2.6007,B 0,C 0,E1 0.1598,E2 -629.9281} C_DIS
LIN {X -4.5567,Y 3.4926,Z 57,A -2.6596,B 0,C 0,E1 0.1598,E2 -629.9283} C_DIS
LIN {X -4.9612,Y 2.8852,Z 57,A -2.7004,B 0,C 0,E1 0.1598,E2 -629.9283} C_DIS
LIN {X -5.2873,Y 2.2325,Z 57,A -2.7401,B 0,C 0,E1 0.1598,E2 -629.9283} C_DIS
LIN {X -5.5282,Y 1.5437,Z 57,A -2.7781,B 0,C 0,E1 0.1598,E2 -629.9283} C_DIS
LIN {X -5.6802,Y 0.8299,Z 57,A -2.814,B 0,C 0,E1 0.1598,E2 -629.9285} C_DIS
LIN {X -5.7373,Y 0.1025,Z 57,A -2.847,B 0,C 0,E1 0.1598,E2 -629.9285} C_DIS
LIN {X -5.7066,Y -0.6266,Z 57,A -2.8768,B 0,C 0,E1 0.1598,E2 -629.9285} C_DIS
LIN {X -5.4737,Y -1.744,Z 57,A -2.9153,B 0,C 0,E1 0.1598,E2 -629.929} C_DIS
LIN {X -5.1143,Y -2.6045,Z 57,A -2.9389,B 0,C 0,E1 0.1598,E2 -629.9287} C_DIS
LIN {X -4.7356,Y -3.2472,Z 57,A -2.9525,B 0,C 0,E1 0.1598,E2 -629.9286} C_DIS
LIN {X -4.2739,Y -3.8332,Z 57,A -2.9604,B 0,C 0,E1 0.1598,E2 -629.9286} C_DIS
LIN {X -3.7391,Y -4.3533,Z 57,A -2.963,B 0,C 0,E1 0.1598,E2 -629.9286} C_DIS
LIN {X -3.1432,Y -4.8016,Z 57,A -2.9602,B 0,C 0,E1 0.1598,E2 -629.9285} C_DIS
LIN {X -2.1239,Y -5.3378,Z 57,A -2.9456,B 0,C 0,E1 0.1598,E2 -629.9285} C_DIS
LIN {X -1.2653,Y -5.598,Z 57,A -2.9253,B 0,C 0,E1 0.1598,E2 -629.9284} C_DIS
LIN {X -0.5569,Y -5.7122,Z 57,A -2.9042,B 0,C 0,E1 0.1598,E2 -629.9284} C_DIS
LIN {X -0.5569,Y -5.7122,Z 57,A -2.9042,B 0,C 0,E1 0.1598,E2 -629.9284} C_DIS
Enddeposition()
LIN {X -0.0081,Y -4.7574,Z 57,A -2.8419,B 0,C 0,E1 0.1598,E2 -629.9296} C_DIS
Startdeposition()
$VEL.CP = VEL_PRINT
LIN {X -0.8144,Y -4.6868,Z 57,A -2.8697,B 0,C 0,E1 0.1598,E2 -629.9283} C_DIS
LIN {X -1.6663,Y -4.454,Z 57,A -2.8911,B 0,C 0,E1 0.1598,E2 -629.9283} C_DIS
LIN {X -2.315,Y -4.1532,Z 57,A -2.9021,B 0,C 0,E1 0.1598,E2 -629.9283} C_DIS
LIN {X -2.9592,Y -3.7232,Z 57,A -2.9074,B 0,C 0,E1 0.1598,E2 -629.9284} C_DIS
LIN {X -3.524,Y -3.1933,Z 57,A -2.9055,B 0,C 0,E1 0.1598,E2 -629.9284} C_DIS
LIN {X -3.9641,Y -2.6296,Z 57,A -2.8977,B 0,C 0,E1 0.1598,E2 -629.9284} C_DIS
LIN {X -4.2861,Y -2.0585,Z 57,A -2.8853,B 0,C 0,E1 0.1598,E2 -629.9284} C_DIS
LIN {X -4.5282,Y -1.4494,Z 57,A -2.8683,B 0,C 0,E1 0.1598,E2 -629.9284} C_DIS
LIN {X -4.7057,Y -0.6955,Z 57,A -2.8426,B 0,C 0,E1 0.1598,E2 -629.9285} C_DIS
LIN {X -4.753,Y 0.1371,Z 57,A -2.809,B 0,C 0,E1 0.1598,E2 -629.9285} C_DIS
LIN {X -4.6876,Y 0.7893,Z 57,A -2.779,B 0,C 0,E1 0.1598,E2 -629.9284} C_DIS
LIN {X -4.5178,Y 1.4838,Z 57,A -2.7432,B 0,C 0,E1 0.1598,E2 -629.9284} C_DIS
LIN {X -4.2181,Y 2.198,Z 57,A -2.7018,B 0,C 0,E1 0.1598,E2 -629.9284} C_DIS
LIN {X -3.8041,Y 2.8526,Z 57,A -2.6589,B 0,C 0,E1 0.1598,E2 -629.9282} C_DIS
LIN {X -3.3704,Y 3.3539,Z 57,A -2.6217,B 0,C 0,E1 0.1598,E2 -629.9281} C_DIS
LIN {X -2.8425,Y 3.8117,Z 57,A -2.5828,B 0,C 0,E1 0.1598,E2 -629.928} C_DIS
LIN {X -2.1296,Y 4.253,Z 57,A -2.5378,B 0,C 0,E1 0.1598,E2 -629.928} C_DIS
LIN {X -1.4164,Y 4.5397,Z 57,A -2.4994,B 0,C 0,E1 0.1598,E2 -629.9278} C_DIS
LIN {X -0.7355,Y 4.6976,Z 57,A -2.4676,B 0,C 0,E1 0.1598,E2 -629.9278} C_DIS
LIN {X 0.0309,Y 4.7561,Z 57,A -2.4369,B 0,C 0,E1 0.1598,E2 -629.9277} C_DIS
LIN {X 0.7965,Y 4.6876,Z 57,A -2.4116,B 0,C 0,E1 0.1598,E2 -629.9277} C_DIS
LIN {X 1.475,Y 4.5201,Z 57,A -2.3937,B 0,C 0,E1 0.1598,E2 -629.9277} C_DIS
LIN {X 2.2468,Y 4.1927,Z 57,A -2.3791,B 0,C 0,E1 0.1598,E2 -629.9277} C_DIS
LIN {X 2.9475,Y 3.7322,Z 57,A -2.3729,B 0,C 0,E1 0.1598,E2 -629.9277} C_DIS
LIN {X 3.5104,Y 3.2087,Z 57,A -2.3744,B 0,C 0,E1 0.1598,E2 -629.9277} C_DIS
LIN {X 3.9822,Y 2.6017,Z 57,A -2.3828,B 0,C 0,E1 0.1598,E2 -629.9278} C_DIS
LIN {X 4.3764,Y 1.8617,Z 57,A -2.3998,B 0,C 0,E1 0.1598,E2 -629.928} C_DIS
LIN {X 4.5947,Y 1.2259,Z 57,A -2.419,B 0,C 0,E1 0.1598,E2 -629.9279} C_DIS
LIN {X 4.7392,Y 0.4068,Z 57,A -2.4485,B 0,C 0,E1 0.1598,E2 -629.9281} C_DIS
LIN {X 4.7358,Y -0.425,Z 57,A -2.4841,B 0,C 0,E1 0.1598,E2 -629.9281} C_DIS
LIN {X 4.6275,Y -1.0922,Z 57,A -2.5167,B 0,C 0,E1 0.1598,E2 -629.9281} C_DIS
LIN {X 4.4277,Y -1.7382,Z 57,A -2.5517,B 0,C 0,E1 0.1598,E2 -629.9281} C_DIS
LIN {X 4.0572,Y -2.483,Z 57,A -2.597,B 0,C 0,E1 0.1598,E2 -629.9281} C_DIS
Enddeposition()
END
